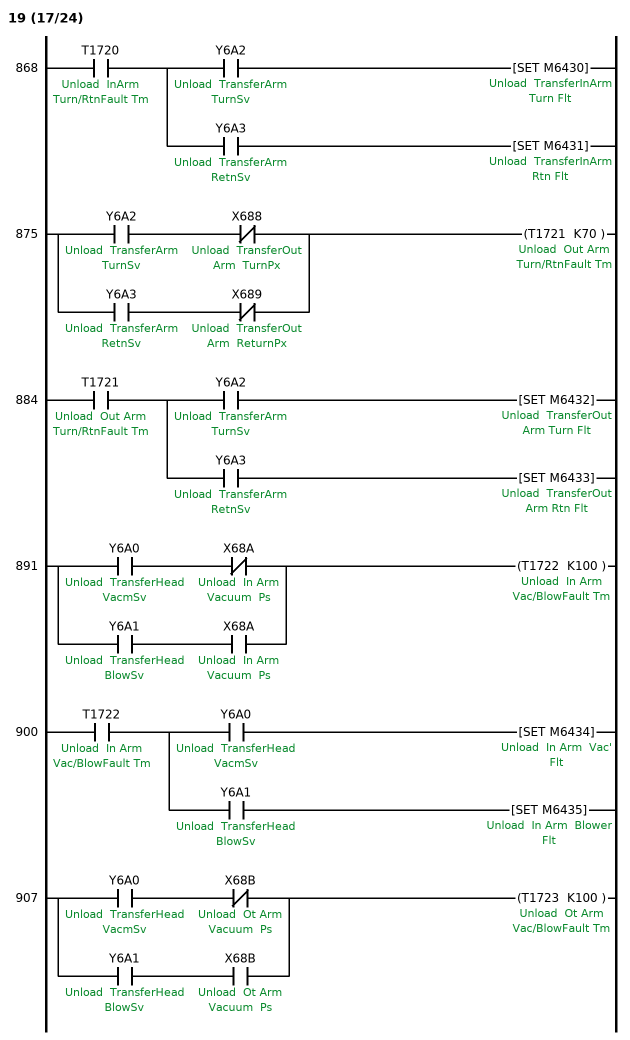
868   LD      T1720  ; Unload  InArm   Turn/RtnFault Tm
      MPS
      AND     Y6A2  ; Unload  TransferArm TurnSv
      SET     M6430  ; Unload  TransferInArm   Turn Flt
      MPP
      AND     Y6A3  ; Unload  TransferArm RetnSv
      SET     M6431  ; Unload  TransferInArm   Rtn Flt
875   LD      Y6A2  ; Unload  TransferArm TurnSv
      ANI     X688  ; Unload  TransferOutArm  TurnPx
      LD      Y6A3  ; Unload  TransferArm RetnSv
      ANI     X689  ; Unload  TransferOutArm  ReturnPx
      ORB
      OUT     T1721 K70  ; Unload  Out Arm Turn/RtnFault Tm
884   LD      T1721  ; Unload  Out Arm Turn/RtnFault Tm
      MPS
      AND     Y6A2  ; Unload  TransferArm TurnSv
      SET     M6432  ; Unload  TransferOut Arm Turn Flt
      MPP
      AND     Y6A3  ; Unload  TransferArm RetnSv
      SET     M6433  ; Unload  TransferOut Arm Rtn Flt
891   LD      Y6A0  ; Unload  TransferHeadVacmSv
      ANI     X68A  ; Unload  In Arm  Vacuum  Ps
      LD      Y6A1  ; Unload  TransferHeadBlowSv
      AND     X68A  ; Unload  In Arm  Vacuum  Ps
      ORB
      OUT     T1722 K100  ; Unload  In Arm  Vac/BlowFault Tm
900   LD      T1722  ; Unload  In Arm  Vac/BlowFault Tm
      MPS
      AND     Y6A0  ; Unload  TransferHeadVacmSv
      SET     M6434  ; Unload  In Arm  Vac' Flt
      MPP
      AND     Y6A1  ; Unload  TransferHeadBlowSv
      SET     M6435  ; Unload  In Arm  Blower  Flt
907   LD      Y6A0  ; Unload  TransferHeadVacmSv
      ANI     X68B  ; Unload  Ot Arm  Vacuum  Ps
      LD      Y6A1  ; Unload  TransferHeadBlowSv
      AND     X68B  ; Unload  Ot Arm  Vacuum  Ps
      ORB
      OUT     T1723 K100  ; Unload  Ot Arm  Vac/BlowFault Tm
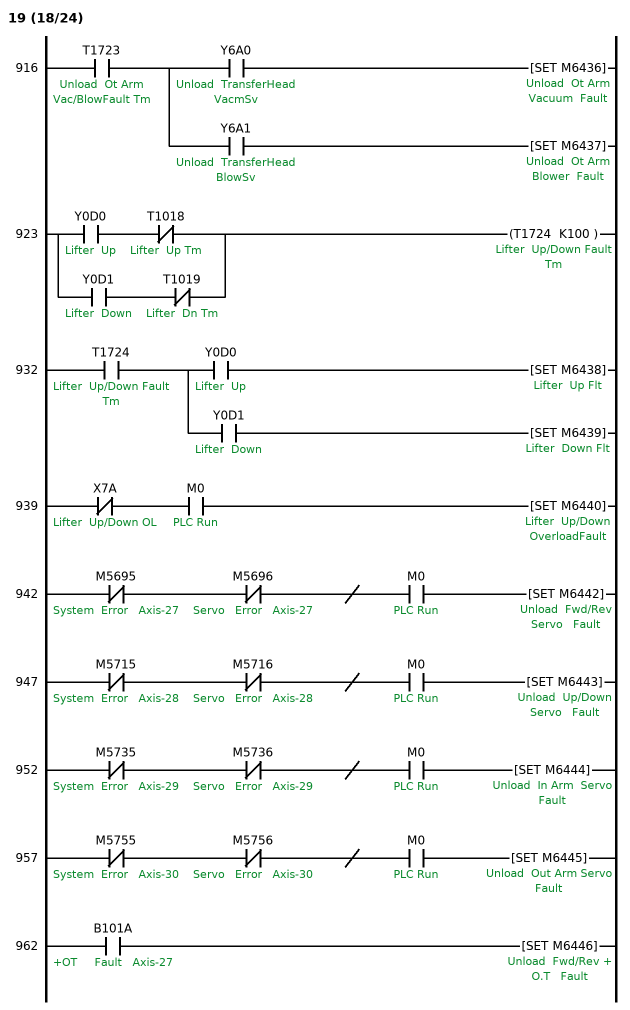
916   LD      T1723  ; Unload  Ot Arm  Vac/BlowFault Tm
      MPS
      AND     Y6A0  ; Unload  TransferHeadVacmSv
      SET     M6436  ; Unload  Ot Arm  Vacuum  Fault
      MPP
      AND     Y6A1  ; Unload  TransferHeadBlowSv
      SET     M6437  ; Unload  Ot Arm  Blower  Fault
923   LD      Y0D0  ; Lifter  Up
      ANI     T1018  ; Lifter  Up Tm
      LD      Y0D1  ; Lifter  Down
      ANI     T1019  ; Lifter  Dn Tm
      ORB
      OUT     T1724 K100  ; Lifter  Up/Down Fault Tm
932   LD      T1724  ; Lifter  Up/Down Fault Tm
      MPS
      AND     Y0D0  ; Lifter  Up
      SET     M6438  ; Lifter  Up Flt
      MPP
      AND     Y0D1  ; Lifter  Down
      SET     M6439  ; Lifter  Down Flt
939   LDI     X7A  ; Lifter  Up/Down OL
      AND     M0  ; PLC Run
      SET     M6440  ; Lifter  Up/Down OverloadFault
942   LDI     M5695  ; System  Error   Axis-27
      ANI     M5696  ; Servo   Error   Axis-27
      INV
      AND     M0  ; PLC Run
      SET     M6442  ; Unload  Fwd/Rev Servo   Fault
947   LDI     M5715  ; System  Error   Axis-28
      ANI     M5716  ; Servo   Error   Axis-28
      INV
      AND     M0  ; PLC Run
      SET     M6443  ; Unload  Up/Down Servo   Fault
952   LDI     M5735  ; System  Error   Axis-29
      ANI     M5736  ; Servo   Error   Axis-29
      INV
      AND     M0  ; PLC Run
      SET     M6444  ; Unload  In Arm  Servo   Fault
957   LDI     M5755  ; System  Error   Axis-30
      ANI     M5756  ; Servo   Error   Axis-30
      INV
      AND     M0  ; PLC Run
      SET     M6445  ; Unload  Out Arm Servo   Fault
962   LD      B101A  ; +OT     Fault   Axis-27
      SET     M6446  ; Unload  Fwd/Rev + O.T   Fault
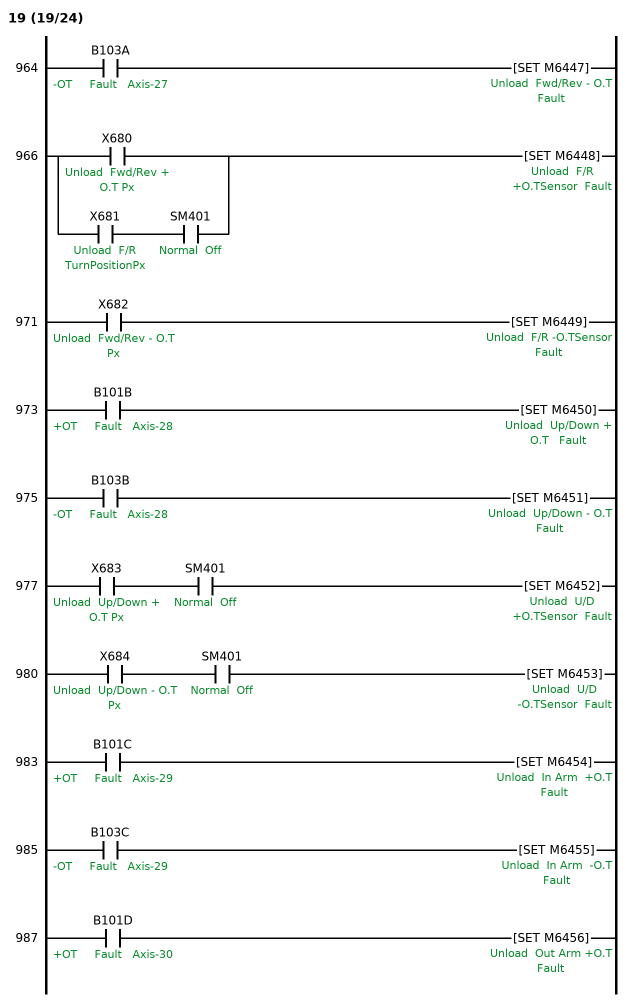
964   LD      B103A  ; -OT     Fault   Axis-27
      SET     M6447  ; Unload  Fwd/Rev - O.T   Fault
966   LD      X680  ; Unload  Fwd/Rev + O.T Px
      LD      X681  ; Unload  F/R TurnPositionPx
      AND     SM401  ; Normal  Off
      ORB
      SET     M6448  ; Unload  F/R +O.TSensor  Fault
971   LD      X682  ; Unload  Fwd/Rev - O.T Px
      SET     M6449  ; Unload  F/R -O.TSensor  Fault
973   LD      B101B  ; +OT     Fault   Axis-28
      SET     M6450  ; Unload  Up/Down + O.T   Fault
975   LD      B103B  ; -OT     Fault   Axis-28
      SET     M6451  ; Unload  Up/Down - O.T   Fault
977   LD      X683  ; Unload  Up/Down + O.T Px
      AND     SM401  ; Normal  Off
      SET     M6452  ; Unload  U/D +O.TSensor  Fault
980   LD      X684  ; Unload  Up/Down - O.T Px
      AND     SM401  ; Normal  Off
      SET     M6453  ; Unload  U/D -O.TSensor  Fault
983   LD      B101C  ; +OT     Fault   Axis-29
      SET     M6454  ; Unload  In Arm  +O.T    Fault
985   LD      B103C  ; -OT     Fault   Axis-29
      SET     M6455  ; Unload  In Arm  -O.T    Fault
987   LD      B101D  ; +OT     Fault   Axis-30
      SET     M6456  ; Unload  Out Arm +O.T    Fault
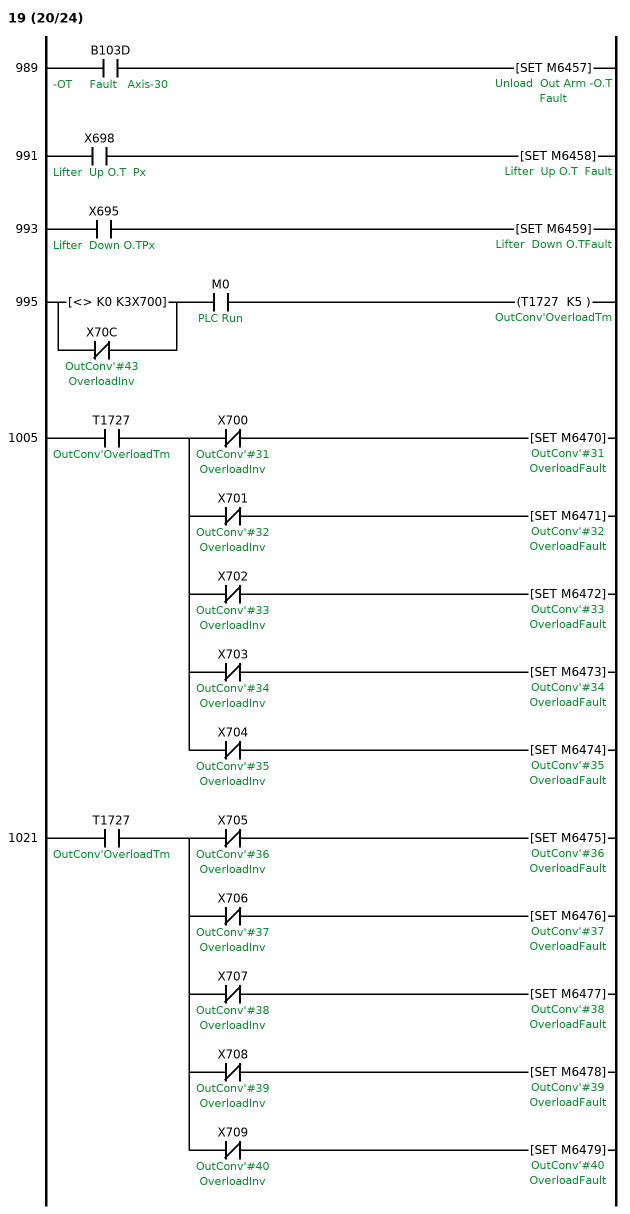
989   LD      B103D  ; -OT     Fault   Axis-30
      SET     M6457  ; Unload  Out Arm -O.T    Fault
991   LD      X698  ; Lifter  Up O.T  Px
      SET     M6458  ; Lifter  Up O.T  Fault
993   LD      X695  ; Lifter  Down O.TPx
      SET     M6459  ; Lifter  Down O.TFault
995   LD<>    K0 K3X700  ; OutConv'#31     OverloadInv
      ORI     X70C  ; OutConv'#43     OverloadInv
      AND     M0  ; PLC Run
      OUT     T1727 K5  ; OutConv'OverloadTm
1005  LD      T1727  ; OutConv'OverloadTm
      MPS
      ANI     X700  ; OutConv'#31     OverloadInv
      SET     M6470  ; OutConv'#31     OverloadFault
      MRD
      ANI     X701  ; OutConv'#32     OverloadInv
      SET     M6471  ; OutConv'#32     OverloadFault
      MRD
      ANI     X702  ; OutConv'#33     OverloadInv
      SET     M6472  ; OutConv'#33     OverloadFault
      MRD
      ANI     X703  ; OutConv'#34     OverloadInv
      SET     M6473  ; OutConv'#34     OverloadFault
      MPP
      ANI     X704  ; OutConv'#35     OverloadInv
      SET     M6474  ; OutConv'#35     OverloadFault
1021  LD      T1727  ; OutConv'OverloadTm
      MPS
      ANI     X705  ; OutConv'#36     OverloadInv
      SET     M6475  ; OutConv'#36     OverloadFault
      MRD
      ANI     X706  ; OutConv'#37     OverloadInv
      SET     M6476  ; OutConv'#37     OverloadFault
      MRD
      ANI     X707  ; OutConv'#38     OverloadInv
      SET     M6477  ; OutConv'#38     OverloadFault
      MRD
      ANI     X708  ; OutConv'#39     OverloadInv
      SET     M6478  ; OutConv'#39     OverloadFault
      MPP
      ANI     X709  ; OutConv'#40     OverloadInv
      SET     M6479  ; OutConv'#40     OverloadFault
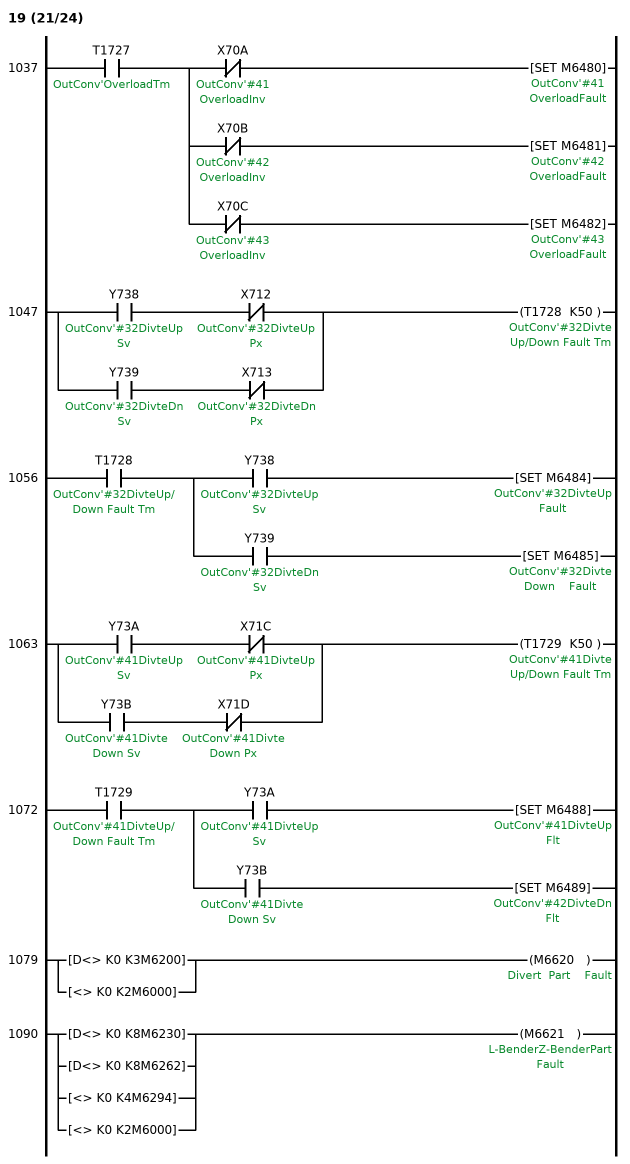
1037  LD      T1727  ; OutConv'OverloadTm
      MPS
      ANI     X70A  ; OutConv'#41     OverloadInv
      SET     M6480  ; OutConv'#41     OverloadFault
      MRD
      ANI     X70B  ; OutConv'#42     OverloadInv
      SET     M6481  ; OutConv'#42     OverloadFault
      MPP
      ANI     X70C  ; OutConv'#43     OverloadInv
      SET     M6482  ; OutConv'#43     OverloadFault
1047  LD      Y738  ; OutConv'#32DivteUp Sv
      ANI     X712  ; OutConv'#32DivteUp Px
      LD      Y739  ; OutConv'#32DivteDn Sv
      ANI     X713  ; OutConv'#32DivteDn Px
      ORB
      OUT     T1728 K50  ; OutConv'#32DivteUp/Down Fault Tm
1056  LD      T1728  ; OutConv'#32DivteUp/Down Fault Tm
      MPS
      AND     Y738  ; OutConv'#32DivteUp Sv
      SET     M6484  ; OutConv'#32DivteUp Fault
      MPP
      AND     Y739  ; OutConv'#32DivteDn Sv
      SET     M6485  ; OutConv'#32DivteDown    Fault
1063  LD      Y73A  ; OutConv'#41DivteUp Sv
      ANI     X71C  ; OutConv'#41DivteUp Px
      LD      Y73B  ; OutConv'#41DivteDown Sv
      ANI     X71D  ; OutConv'#41DivteDown Px
      ORB
      OUT     T1729 K50  ; OutConv'#41DivteUp/Down Fault Tm
1072  LD      T1729  ; OutConv'#41DivteUp/Down Fault Tm
      MPS
      AND     Y73A  ; OutConv'#41DivteUp Sv
      SET     M6488  ; OutConv'#41DivteUp Flt
      MPP
      AND     Y73B  ; OutConv'#41DivteDown Sv
      SET     M6489  ; OutConv'#42DivteDn Flt
1079  LDD<>   K0 K3M6200  ; Divert#1In Conv'OL Fault
      OR<>    K0 K2M6000  ; Emg-StopFault
      OUT     M6620  ; Divert  Part    Fault
1090  LDD<>   K0 K8M6230  ; Z-BendInClamp UpFault
      ORD<>   K0 K8M6262  ; Z-Bend  Conv' UpFault
      OR<>    K0 K4M6294  ; Z-BendInServo   Fault
      OR<>    K0 K2M6000  ; Emg-StopFault
      OUT     M6621  ; L-BenderZ-BenderPart    Fault
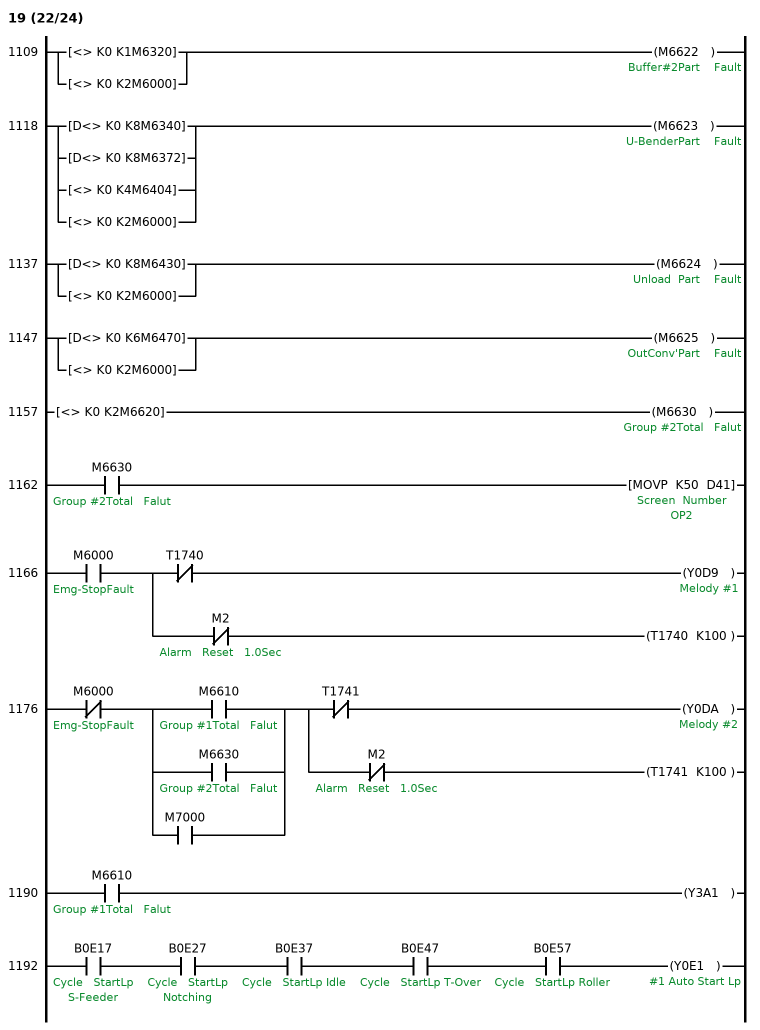
1109  LD<>    K0 K1M6320  ; Buffer#2ConveyorConv' OLFault
      OR<>    K0 K2M6000  ; Emg-StopFault
      OUT     M6622  ; Buffer#2Part    Fault
1118  LDD<>   K0 K8M6340  ; U-BenderConv' OLFalut
      ORD<>   K0 K8M6372  ; U-BendOtUpper   Guide   FwdFault
      OR<>    K0 K4M6404  ; U-BendOtLength  Unit    +O.TFlt
      OR<>    K0 K2M6000  ; Emg-StopFault
      OUT     M6623  ; U-BenderPart    Fault
1137  LDD<>   K0 K8M6430  ; Unload  TransferInArm   Turn Flt
      OR<>    K0 K2M6000  ; Emg-StopFault
      OUT     M6624  ; Unload  Part    Fault
1147  LDD<>   K0 K6M6470  ; OutConv'#31     OverloadFault
      OR<>    K0 K2M6000  ; Emg-StopFault
      OUT     M6625  ; OutConv'Part    Fault
1157  LD<>    K0 K2M6620  ; Divert  Part    Fault
      OUT     M6630  ; Group #2Total   Falut
1162  LD      M6630  ; Group #2Total   Falut
      MOVP    K50 D41  ; Screen  Number  OP2
1166  LD      M6000  ; Emg-StopFault
      MPS
      ANI     T1740
      OUT     Y0D9  ; Melody #1
      MPP
      ANI     M2  ; Alarm   Reset   1.0Sec
      OUT     T1740 K100
1176  LDI     M6000  ; Emg-StopFault
      LD      M6610  ; Group #1Total   Falut
      OR      M6630  ; Group #2Total   Falut
      OR      M7000
      ANB
      MPS
      ANI     T1741
      OUT     Y0DA  ; Melody #2
      MPP
      ANI     M2  ; Alarm   Reset   1.0Sec
      OUT     T1741 K100
1190  LD      M6610  ; Group #1Total   Falut
      OUT     Y3A1
1192  LD      B0E17  ; Cycle   StartLp S-Feeder
      AND     B0E27  ; Cycle   StartLp Notching
      AND     B0E37  ; Cycle   StartLp Idle
      AND     B0E47  ; Cycle   StartLp T-Over
      AND     B0E57  ; Cycle   StartLp Roller
      OUT     Y0E1  ; #1 Auto Start Lp
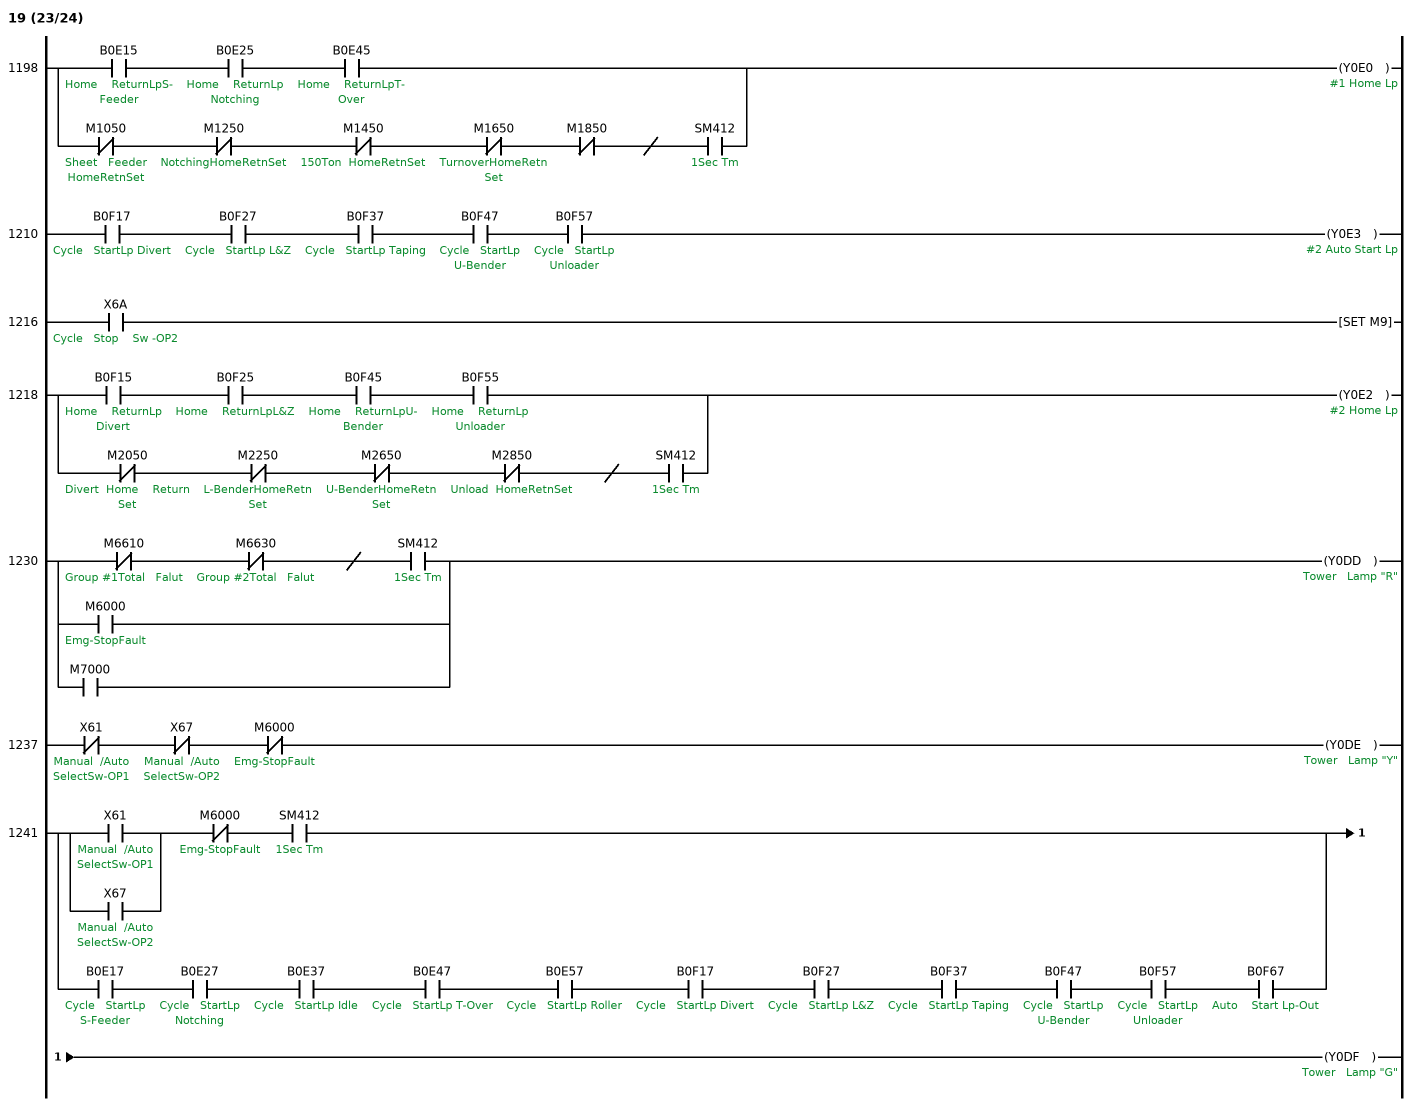
1198  LD      B0E15  ; Home    ReturnLpS-Feeder
      AND     B0E25  ; Home    ReturnLpNotching
      AND     B0E45  ; Home    ReturnLpT-Over
      LDI     M1050  ; Sheet   Feeder  HomeRetnSet
      ANI     M1250  ; NotchingHomeRetnSet
      ANI     M1450  ; 150Ton  HomeRetnSet
      ANI     M1650  ; TurnoverHomeRetnSet
      ANI     M1850
      INV
      AND     SM412  ; 1Sec Tm
      ORB
      OUT     Y0E0  ; #1 Home Lp
1210  LD      B0F17  ; Cycle   StartLp Divert
      AND     B0F27  ; Cycle   StartLp L&Z
      AND     B0F37  ; Cycle   StartLp Taping
      AND     B0F47  ; Cycle   StartLp U-Bender
      AND     B0F57  ; Cycle   StartLp Unloader
      OUT     Y0E3  ; #2 Auto Start Lp
1216  LD      X6A  ; Cycle   Stop    Sw -OP2
      SET     M9
1218  LD      B0F15  ; Home    ReturnLpDivert
      AND     B0F25  ; Home    ReturnLpL&Z
      AND     B0F45  ; Home    ReturnLpU-Bender
      AND     B0F55  ; Home    ReturnLpUnloader
      LDI     M2050  ; Divert  Home    Return  Set
      ANI     M2250  ; L-BenderHomeRetnSet
      ANI     M2650  ; U-BenderHomeRetnSet
      ANI     M2850  ; Unload  HomeRetnSet
      INV
      AND     SM412  ; 1Sec Tm
      ORB
      OUT     Y0E2  ; #2 Home Lp
1230  LDI     M6610  ; Group #1Total   Falut
      ANI     M6630  ; Group #2Total   Falut
      INV
      AND     SM412  ; 1Sec Tm
      OR      M6000  ; Emg-StopFault
      OR      M7000
      OUT     Y0DD  ; Tower   Lamp "R"
1237  LDI     X61  ; Manual  /Auto   SelectSw-OP1
      ANI     X67  ; Manual  /Auto   SelectSw-OP2
      ANI     M6000  ; Emg-StopFault
      OUT     Y0DE  ; Tower   Lamp "Y"
1241  LD      X61  ; Manual  /Auto   SelectSw-OP1
      OR      X67  ; Manual  /Auto   SelectSw-OP2
      ANI     M6000  ; Emg-StopFault
      AND     SM412  ; 1Sec Tm
      LD      B0E17  ; Cycle   StartLp S-Feeder
      AND     B0E27  ; Cycle   StartLp Notching
      AND     B0E37  ; Cycle   StartLp Idle
      AND     B0E47  ; Cycle   StartLp T-Over
      AND     B0E57  ; Cycle   StartLp Roller
      AND     B0F17  ; Cycle   StartLp Divert
      AND     B0F27  ; Cycle   StartLp L&Z
      AND     B0F37  ; Cycle   StartLp Taping
      AND     B0F47  ; Cycle   StartLp U-Bender
      AND     B0F57  ; Cycle   StartLp Unloader
      AND     B0F67  ; Auto    Start Lp-Out
      ORB
      OUT     Y0DF  ; Tower   Lamp "G"
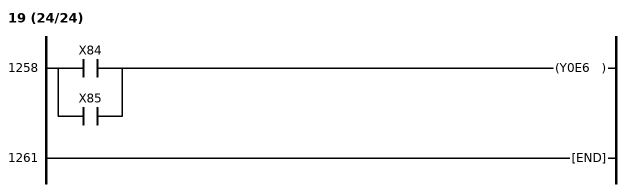
1258  LD      X84
      OR      X85
      OUT     Y0E6
1261  END
END_PROGRAM

PROGRAM 20  // #2 Conveyor Part
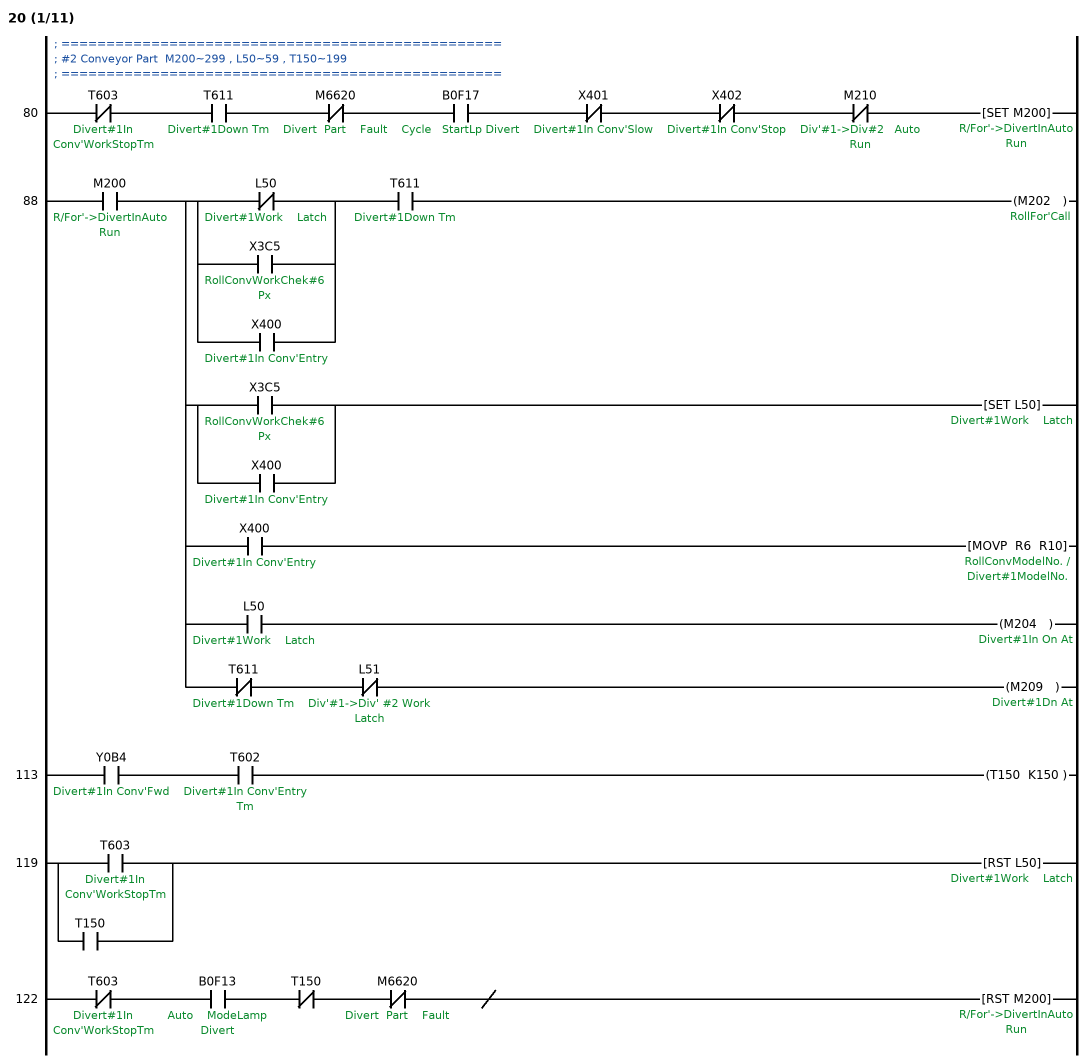
; =================================================
; #2 Conveyor Part  M200~299 , L50~59 , T150~199
; =================================================
80    LDI     T603  ; Divert#1In Conv'WorkStopTm
      AND     T611  ; Divert#1Down Tm
      ANI     M6620  ; Divert  Part    Fault
      AND     B0F17  ; Cycle   StartLp Divert
      ANI     X401  ; Divert#1In Conv'Slow
      ANI     X402  ; Divert#1In Conv'Stop
      ANI     M210  ; Div'#1->Div#2   Auto Run
      SET     M200  ; R/For'->DivertInAuto Run
88    LD      M200  ; R/For'->DivertInAuto Run
      MPS
      LDI     L50  ; Divert#1Work    Latch
      OR      X3C5  ; RollConvWorkChek#6 Px
      OR      X400  ; Divert#1In Conv'Entry
      ANB
      AND     T611  ; Divert#1Down Tm
      OUT     M202  ; RollFor'Call
      MRD
      LD      X3C5  ; RollConvWorkChek#6 Px
      OR      X400  ; Divert#1In Conv'Entry
      ANB
      SET     L50  ; Divert#1Work    Latch
      MRD
      AND     X400  ; Divert#1In Conv'Entry
      MOVP    R6 R10  ; RollConvModelNo. / Divert#1ModelNo.
      MRD
      AND     L50  ; Divert#1Work    Latch
      OUT     M204  ; Divert#1In On At
      MPP
      ANI     T611  ; Divert#1Down Tm
      ANI     L51  ; Div'#1->Div' #2 Work    Latch
      OUT     M209  ; Divert#1Dn At
113   LD      Y0B4  ; Divert#1In Conv'Fwd
      AND     T602  ; Divert#1In Conv'Entry Tm
      OUT     T150 K150
119   LD      T603  ; Divert#1In Conv'WorkStopTm
      OR      T150
      RST     L50  ; Divert#1Work    Latch
122   LDI     T603  ; Divert#1In Conv'WorkStopTm
      AND     B0F13  ; Auto    ModeLampDivert
      ANI     T150
      ANI     M6620  ; Divert  Part    Fault
      INV
      RST     M200  ; R/For'->DivertInAuto Run
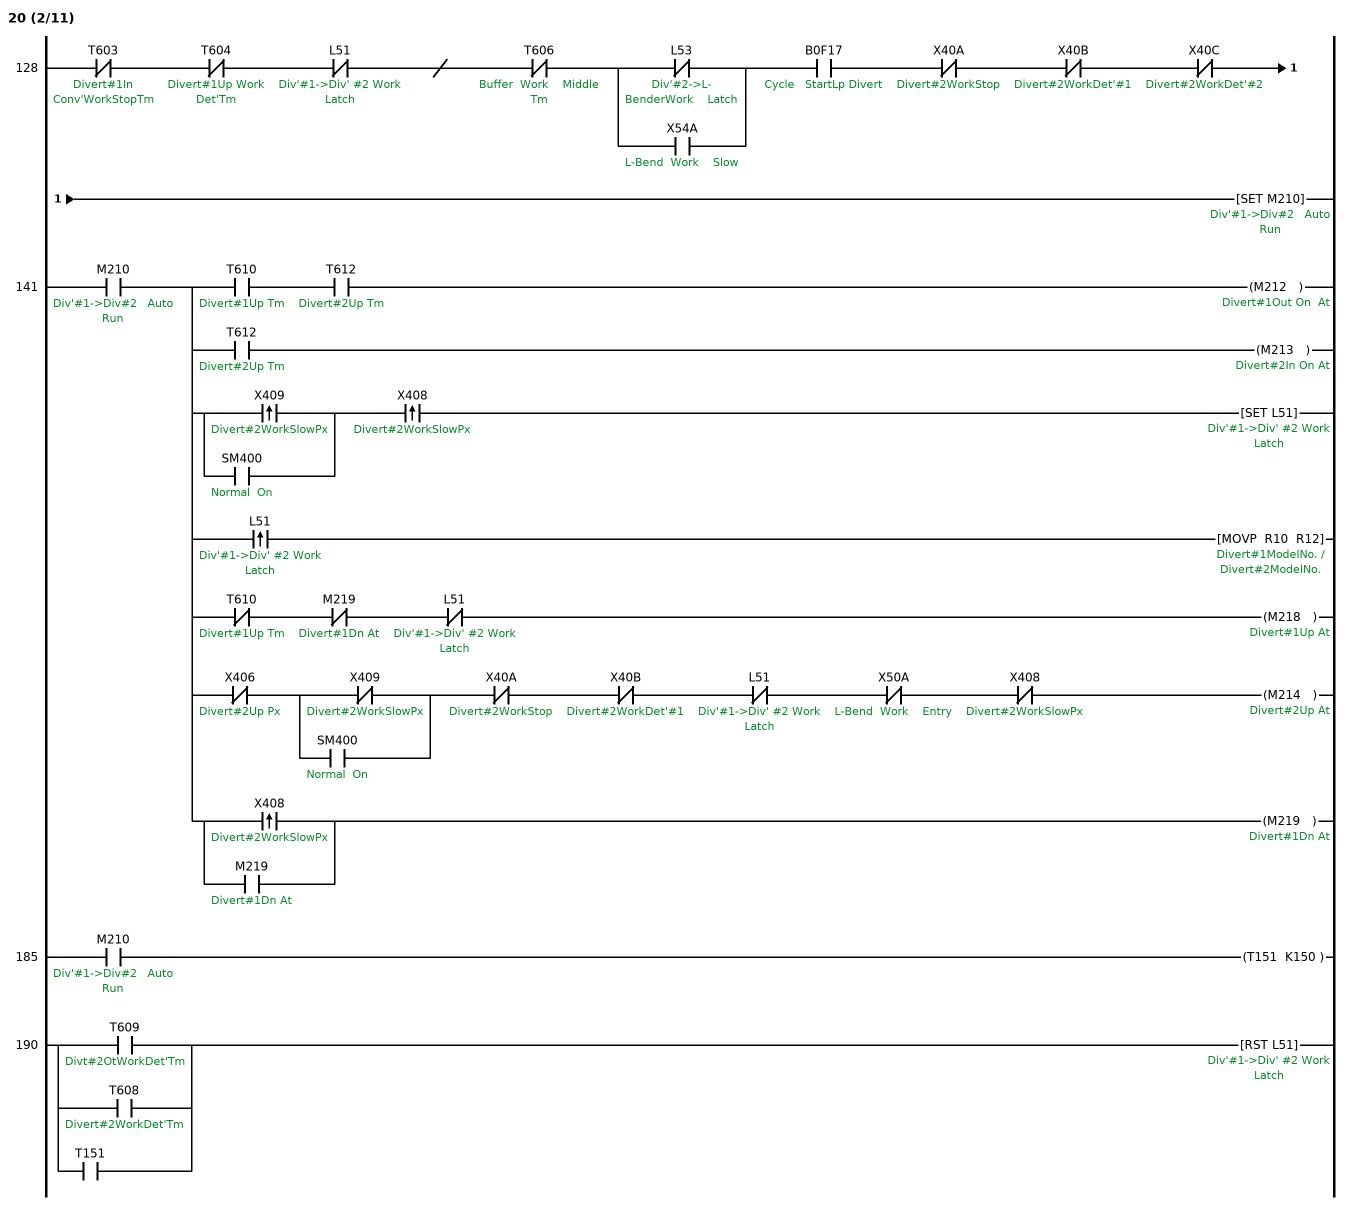
128   LDI     T603  ; Divert#1In Conv'WorkStopTm
      ANI     T604  ; Divert#1Up Work Det'Tm
      ANI     L51  ; Div'#1->Div' #2 Work    Latch
      INV
      ANI     T606  ; Buffer  Work    Middle  Tm
      LDI     L53  ; Div'#2->L-BenderWork    Latch
      OR      X54A  ; L-Bend  Work    Slow
      ANB
      AND     B0F17  ; Cycle   StartLp Divert
      ANI     X40A  ; Divert#2WorkStop
      ANI     X40B  ; Divert#2WorkDet'#1
      ANI     X40C  ; Divert#2WorkDet'#2
      SET     M210  ; Div'#1->Div#2   Auto Run
141   LD      M210  ; Div'#1->Div#2   Auto Run
      MPS
      AND     T610  ; Divert#1Up Tm
      AND     T612  ; Divert#2Up Tm
      OUT     M212  ; Divert#1Out On  At
      MRD
      AND     T612  ; Divert#2Up Tm
      OUT     M213  ; Divert#2In On At
      MRD
      LDP     X409  ; Divert#2WorkSlowPx
      OR      SM400  ; Normal  On
      ANB
      ANDP    X408  ; Divert#2WorkSlowPx
      SET     L51  ; Div'#1->Div' #2 Work    Latch
      MRD
      ANDP    L51  ; Div'#1->Div' #2 Work    Latch
      MOVP    R10 R12  ; Divert#2ModelNo.
      MRD
      ANI     T610  ; Divert#1Up Tm
      ANI     M219  ; Divert#1Dn At
      ANI     L51  ; Div'#1->Div' #2 Work    Latch
      OUT     M218  ; Divert#1Up At
      MRD
      ANI     X406  ; Divert#2Up Px
      LDI     X409  ; Divert#2WorkSlowPx
      OR      SM400  ; Normal  On
      ANB
      ANI     X40A  ; Divert#2WorkStop
      ANI     X40B  ; Divert#2WorkDet'#1
      ANI     L51  ; Div'#1->Div' #2 Work    Latch
      ANI     X50A  ; L-Bend  Work    Entry
      ANI     X408  ; Divert#2WorkSlowPx
      OUT     M214  ; Divert#2Up At
      MPP
      LDP     X408  ; Divert#2WorkSlowPx
      OR      M219  ; Divert#1Dn At
      ANB
      OUT     M219  ; Divert#1Dn At
185   LD      M210  ; Div'#1->Div#2   Auto Run
      OUT     T151 K150
190   LD      T609  ; Divt#2OtWorkDet'Tm
      OR      T608  ; Divert#2WorkDet'Tm
      OR      T151
      RST     L51  ; Div'#1->Div' #2 Work    Latch
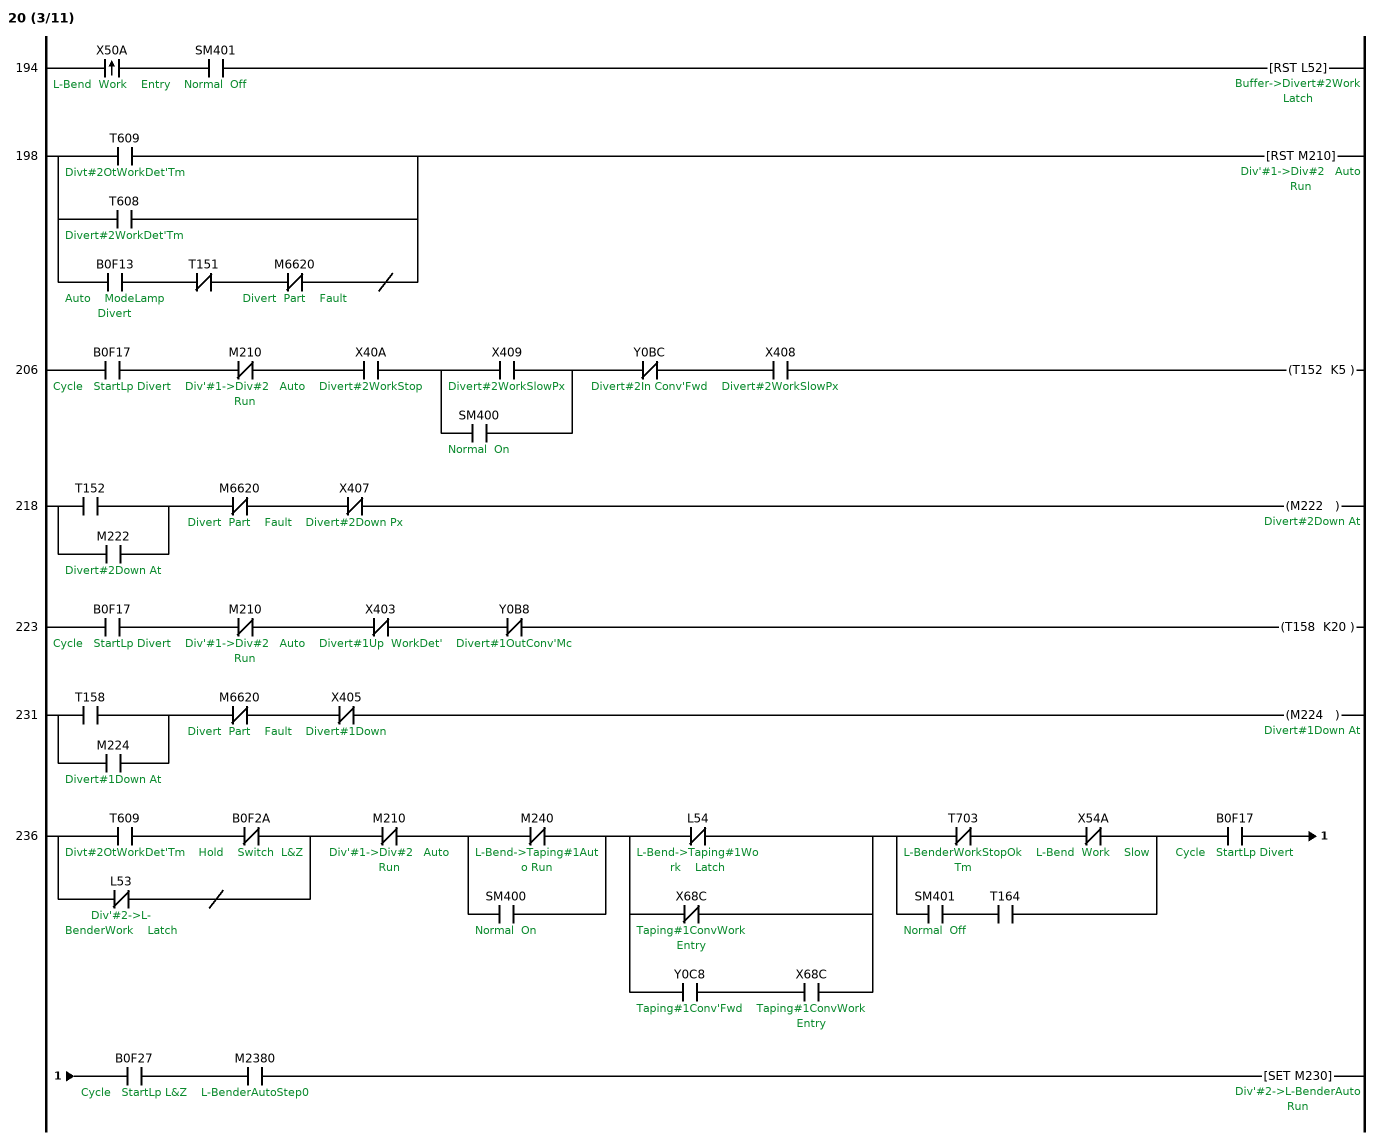
194   LDP     X50A  ; L-Bend  Work    Entry
      AND     SM401  ; Normal  Off
      RST     L52  ; Buffer->Divert#2Work    Latch
198   LD      T609  ; Divt#2OtWorkDet'Tm
      OR      T608  ; Divert#2WorkDet'Tm
      LD      B0F13  ; Auto    ModeLampDivert
      ANI     T151
      ANI     M6620  ; Divert  Part    Fault
      INV
      ORB
      RST     M210  ; Div'#1->Div#2   Auto Run
206   LD      B0F17  ; Cycle   StartLp Divert
      ANI     M210  ; Div'#1->Div#2   Auto Run
      AND     X40A  ; Divert#2WorkStop
      LD      X409  ; Divert#2WorkSlowPx
      OR      SM400  ; Normal  On
      ANB
      ANI     Y0BC  ; Divert#2In Conv'Fwd
      AND     X408  ; Divert#2WorkSlowPx
      OUT     T152 K5
218   LD      T152
      OR      M222  ; Divert#2Down At
      ANI     M6620  ; Divert  Part    Fault
      ANI     X407  ; Divert#2Down Px
      OUT     M222  ; Divert#2Down At
223   LD      B0F17  ; Cycle   StartLp Divert
      ANI     M210  ; Div'#1->Div#2   Auto Run
      ANI     X403  ; Divert#1Up  WorkDet'
      ANI     Y0B8  ; Divert#1OutConv'Mc
      OUT     T158 K20
231   LD      T158
      OR      M224  ; Divert#1Down At
      ANI     M6620  ; Divert  Part    Fault
      ANI     X405  ; Divert#1Down
      OUT     M224  ; Divert#1Down At
236   LD      T609  ; Divt#2OtWorkDet'Tm
      ANI     B0F2A  ; Hold    Switch  L&Z
      LDI     L53  ; Div'#2->L-BenderWork    Latch
      INV
      ORB
      ANI     M210  ; Div'#1->Div#2   Auto Run
      LDI     M240  ; L-Bend->Taping#1Auto Run
      OR      SM400  ; Normal  On
      ANB
      LDI     L54  ; L-Bend->Taping#1Work    Latch
      ORI     X68C  ; Taping#1ConvWorkEntry
      LD      Y0C8  ; Taping#1Conv'Fwd
      AND     X68C  ; Taping#1ConvWorkEntry
      ORB
      ANB
      LDI     T703  ; L-BenderWorkStopOk Tm
      ANI     X54A  ; L-Bend  Work    Slow
      LD      SM401  ; Normal  Off
      AND     T164
      ORB
      ANB
      AND     B0F17  ; Cycle   StartLp Divert
      AND     B0F27  ; Cycle   StartLp L&Z
      AND     M2380  ; L-BenderAutoStep0
      SET     M230  ; Div'#2->L-BenderAuto Run
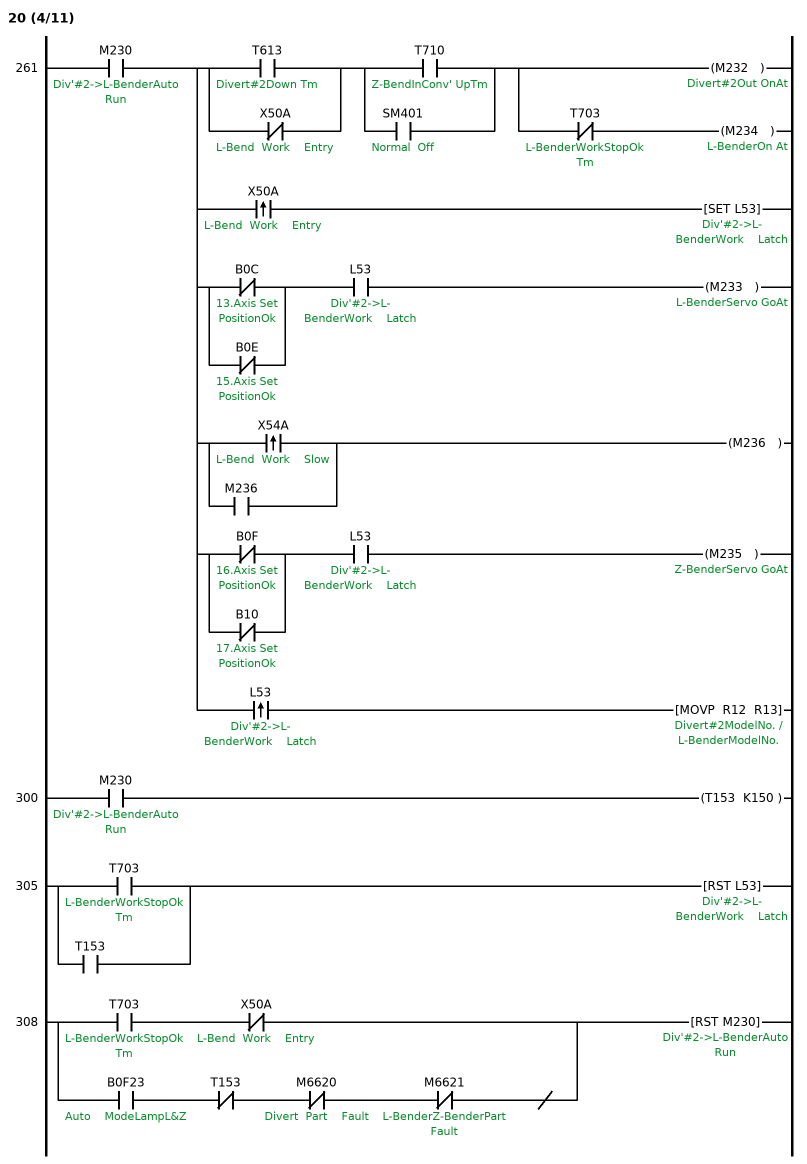
261   LD      M230  ; Div'#2->L-BenderAuto Run
      MPS
      LD      T613  ; Divert#2Down Tm
      ORI     X50A  ; L-Bend  Work    Entry
      ANB
      LD      T710  ; Z-BendInConv' UpTm
      OR      SM401  ; Normal  Off
      ANB
      OUT     M232  ; Divert#2Out OnAt
      ANI     T703  ; L-BenderWorkStopOk Tm
      OUT     M234  ; L-BenderOn At
      MRD
      ANDP    X50A  ; L-Bend  Work    Entry
      SET     L53  ; Div'#2->L-BenderWork    Latch
      MRD
      LDI     B0C  ; 13.Axis Set     PositionOk
      ORI     B0E  ; 15.Axis Set     PositionOk
      ANB
      AND     L53  ; Div'#2->L-BenderWork    Latch
      OUT     M233  ; L-BenderServo GoAt
      MRD
      LDP     X54A  ; L-Bend  Work    Slow
      OR      M236
      ANB
      OUT     M236
      MRD
      LDI     B0F  ; 16.Axis Set     PositionOk
      ORI     B10  ; 17.Axis Set     PositionOk
      ANB
      AND     L53  ; Div'#2->L-BenderWork    Latch
      OUT     M235  ; Z-BenderServo GoAt
      MPP
      ANDP    L53  ; Div'#2->L-BenderWork    Latch
      MOVP    R12 R13  ; L-BenderModelNo.
300   LD      M230  ; Div'#2->L-BenderAuto Run
      OUT     T153 K150
305   LD      T703  ; L-BenderWorkStopOk Tm
      OR      T153
      RST     L53  ; Div'#2->L-BenderWork    Latch
308   LD      T703  ; L-BenderWorkStopOk Tm
      ANI     X50A  ; L-Bend  Work    Entry
      LD      B0F23  ; Auto    ModeLampL&Z
      ANI     T153
      ANI     M6620  ; Divert  Part    Fault
      ANI     M6621  ; L-BenderZ-BenderPart    Fault
      INV
      ORB
      RST     M230  ; Div'#2->L-BenderAuto Run
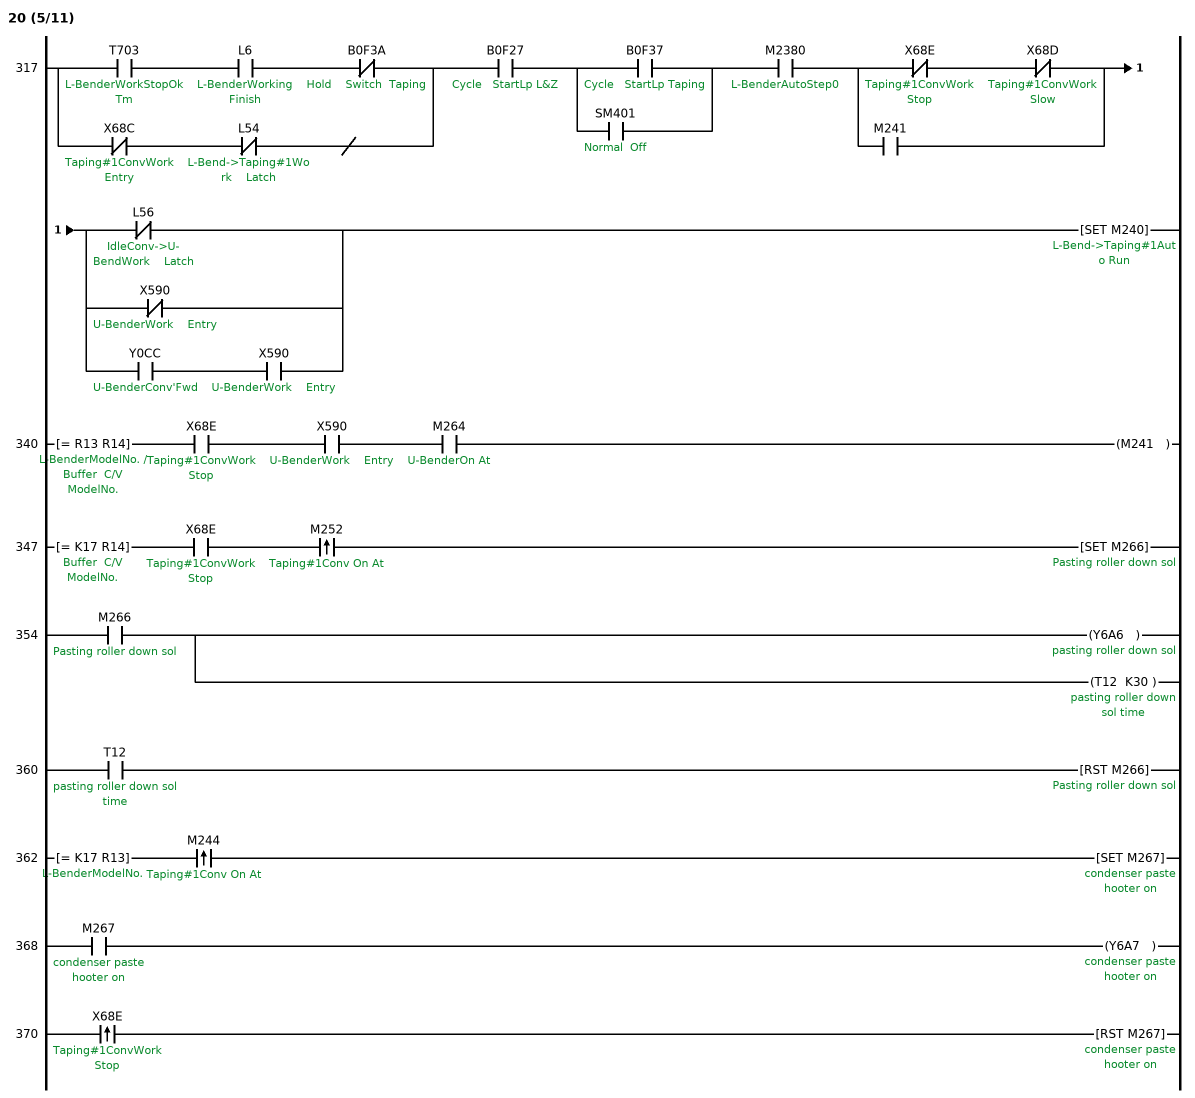
317   LD      T703  ; L-BenderWorkStopOk Tm
      AND     L6  ; L-BenderWorking Finish
      ANI     B0F3A  ; Hold    Switch  Taping
      LDI     X68C  ; Taping#1ConvWorkEntry
      ANI     L54  ; L-Bend->Taping#1Work    Latch
      INV
      ORB
      AND     B0F27  ; Cycle   StartLp L&Z
      LD      B0F37  ; Cycle   StartLp Taping
      OR      SM401  ; Normal  Off
      ANB
      AND     M2380  ; L-BenderAutoStep0
      LDI     X68E  ; Taping#1ConvWorkStop
      ANI     X68D  ; Taping#1ConvWorkSlow
      OR      M241
      ANB
      LDI     L56  ; IdleConv->U-BendWork    Latch
      ORI     X590  ; U-BenderWork    Entry
      LD      Y0CC  ; U-BenderConv'Fwd
      AND     X590  ; U-BenderWork    Entry
      ORB
      ANB
      SET     M240  ; L-Bend->Taping#1Auto Run
340   LD=     R13 R14  ; L-BenderModelNo. / Buffer  C/V     ModelNo.
      AND     X68E  ; Taping#1ConvWorkStop
      AND     X590  ; U-BenderWork    Entry
      AND     M264  ; U-BenderOn At
      OUT     M241
347   LD=     K17 R14  ; Buffer  C/V     ModelNo.
      AND     X68E  ; Taping#1ConvWorkStop
      ANDP    M252  ; Taping#1Conv On At
      SET     M266  ; Pasting roller down sol
354   LD      M266  ; Pasting roller down sol
      OUT     Y6A6  ; pasting roller down sol
      OUT     T12 K30  ; pasting roller down sol time
360   LD      T12  ; pasting roller down sol time
      RST     M266  ; Pasting roller down sol
362   LD=     K17 R13  ; L-BenderModelNo.
      ANDP    M244  ; Taping#1Conv On At
      SET     M267  ; condenser paste hooter on
368   LD      M267  ; condenser paste hooter on
      OUT     Y6A7  ; condenser paste hooter on
370   LDP     X68E  ; Taping#1ConvWorkStop
      RST     M267  ; condenser paste hooter on
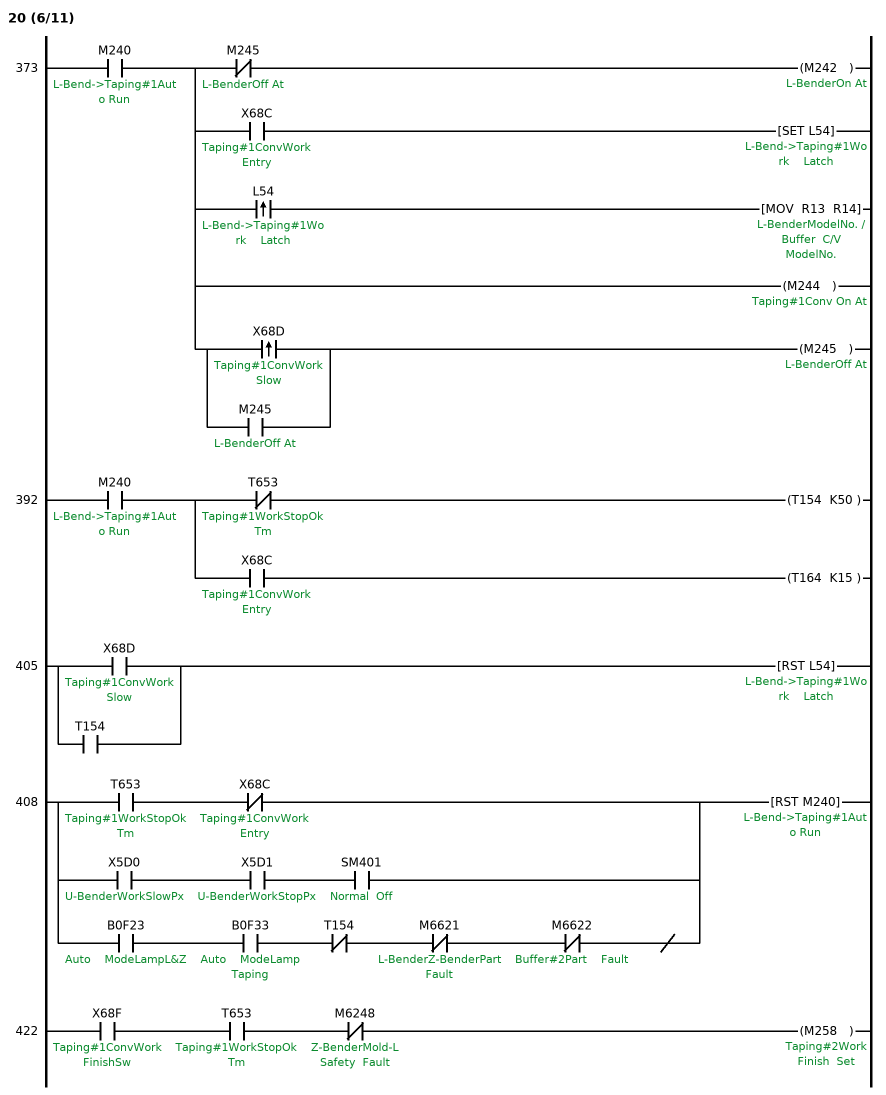
373   LD      M240  ; L-Bend->Taping#1Auto Run
      MPS
      ANI     M245  ; L-BenderOff At
      OUT     M242  ; L-BenderOn At
      MRD
      AND     X68C  ; Taping#1ConvWorkEntry
      SET     L54  ; L-Bend->Taping#1Work    Latch
      MRD
      ANDP    L54  ; L-Bend->Taping#1Work    Latch
      MOV     R13 R14
      MPP
      OUT     M244  ; Taping#1Conv On At
      LDP     X68D  ; Taping#1ConvWorkSlow
      OR      M245  ; L-BenderOff At
      ANB
      OUT     M245  ; L-BenderOff At
392   LD      M240  ; L-Bend->Taping#1Auto Run
      MPS
      ANI     T653  ; Taping#1WorkStopOk Tm
      OUT     T154 K50
      MPP
      AND     X68C  ; Taping#1ConvWorkEntry
      OUT     T164 K15
405   LD      X68D  ; Taping#1ConvWorkSlow
      OR      T154
      RST     L54  ; L-Bend->Taping#1Work    Latch
408   LD      T653  ; Taping#1WorkStopOk Tm
      ANI     X68C  ; Taping#1ConvWorkEntry
      LD      X5D0  ; U-BenderWorkSlowPx
      AND     X5D1  ; U-BenderWorkStopPx
      AND     SM401  ; Normal  Off
      ORB
      LD      B0F23  ; Auto    ModeLampL&Z
      AND     B0F33  ; Auto    ModeLampTaping
      ANI     T154
      ANI     M6621  ; L-BenderZ-BenderPart    Fault
      ANI     M6622  ; Buffer#2Part    Fault
      INV
      ORB
      RST     M240  ; L-Bend->Taping#1Auto Run
422   LD      X68F  ; Taping#1ConvWorkFinishSw
      AND     T653  ; Taping#1WorkStopOk Tm
      ANI     M6248  ; Z-BenderMold-L  Safety  Fault
      OUT     M258  ; Taping#2Work    Finish  Set
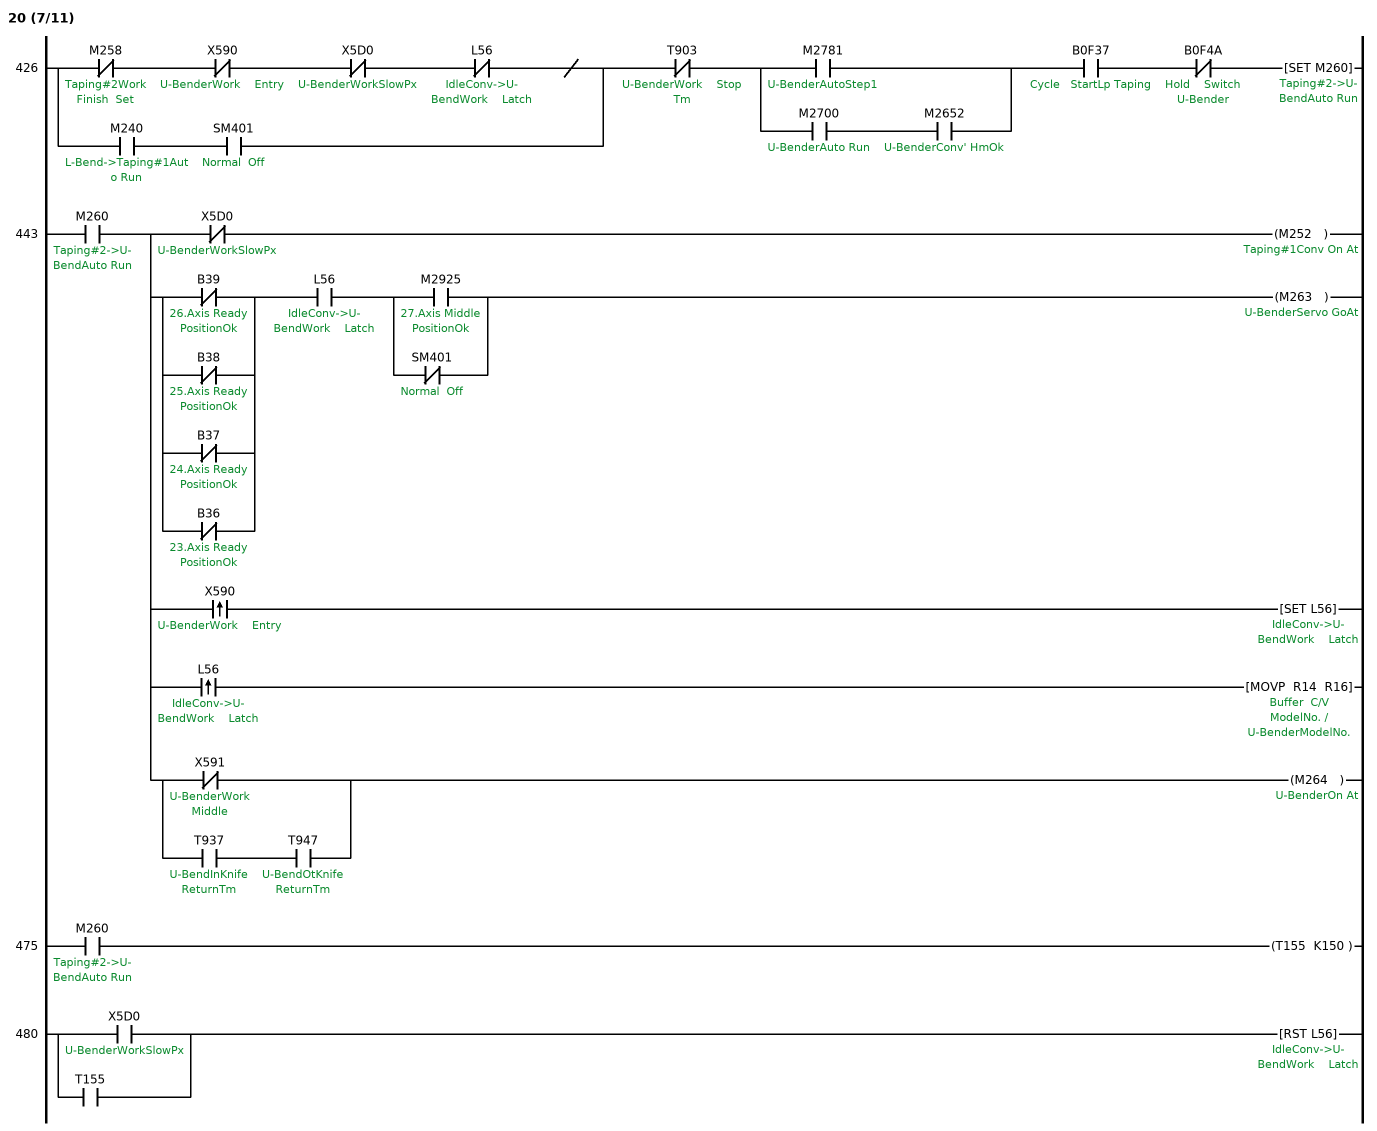
426   LDI     M258  ; Taping#2Work    Finish  Set
      ANI     X590  ; U-BenderWork    Entry
      ANI     X5D0  ; U-BenderWorkSlowPx
      ANI     L56  ; IdleConv->U-BendWork    Latch
      INV
      LD      M240  ; L-Bend->Taping#1Auto Run
      AND     SM401  ; Normal  Off
      ORB
      ANI     T903  ; U-BenderWork    Stop Tm
      LD      M2781  ; U-BenderAutoStep1
      LD      M2700  ; U-BenderAuto Run
      AND     M2652  ; U-BenderConv' HmOk
      ORB
      ANB
      AND     B0F37  ; Cycle   StartLp Taping
      ANI     B0F4A  ; Hold    Switch  U-Bender
      SET     M260  ; Taping#2->U-BendAuto Run
443   LD      M260  ; Taping#2->U-BendAuto Run
      MPS
      ANI     X5D0  ; U-BenderWorkSlowPx
      OUT     M252  ; Taping#1Conv On At
      MRD
      LDI     B39  ; 26.Axis Ready   PositionOk
      ORI     B38  ; 25.Axis Ready   PositionOk
      ORI     B37  ; 24.Axis Ready   PositionOk
      ORI     B36  ; 23.Axis Ready   PositionOk
      ANB
      AND     L56  ; IdleConv->U-BendWork    Latch
      LD      M2925  ; 27.Axis Middle  PositionOk
      ORI     SM401  ; Normal  Off
      ANB
      OUT     M263  ; U-BenderServo GoAt
      MRD
      ANDP    X590  ; U-BenderWork    Entry
      SET     L56  ; IdleConv->U-BendWork    Latch
      MRD
      ANDP    L56  ; IdleConv->U-BendWork    Latch
      MOVP    R14 R16  ; U-BenderModelNo.
      MPP
      LDI     X591  ; U-BenderWork    Middle
      LD      T937  ; U-BendInKnife   ReturnTm
      AND     T947  ; U-BendOtKnife   ReturnTm
      ORB
      ANB
      OUT     M264  ; U-BenderOn At
475   LD      M260  ; Taping#2->U-BendAuto Run
      OUT     T155 K150
480   LD      X5D0  ; U-BenderWorkSlowPx
      OR      T155
      RST     L56  ; IdleConv->U-BendWork    Latch
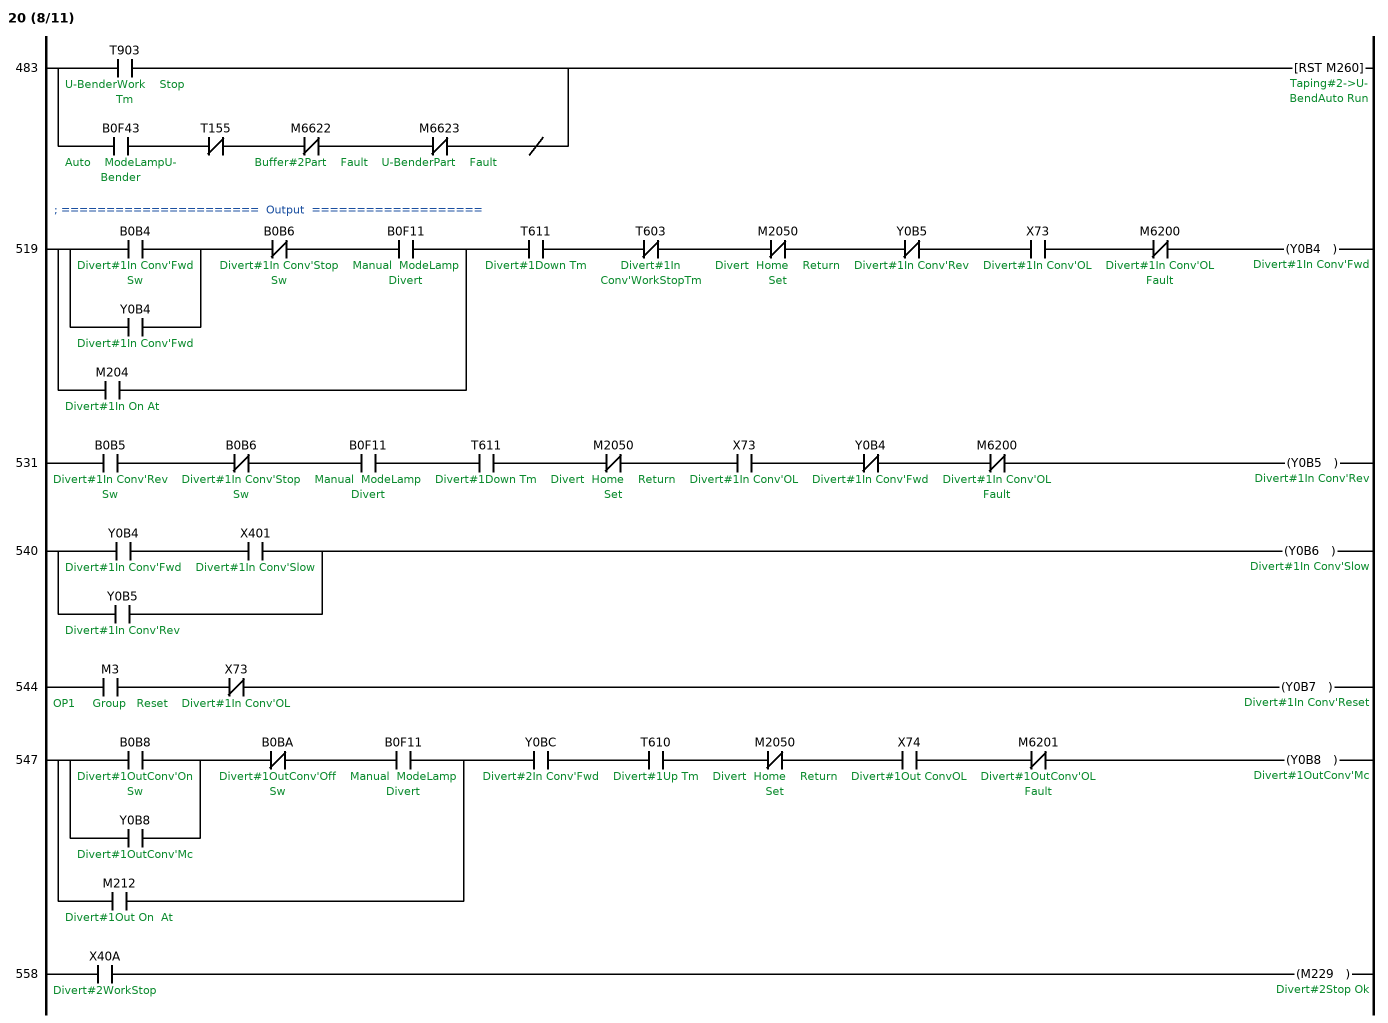
483   LD      T903  ; U-BenderWork    Stop Tm
      LD      B0F43  ; Auto    ModeLampU-Bender
      ANI     T155
      ANI     M6622  ; Buffer#2Part    Fault
      ANI     M6623  ; U-BenderPart    Fault
      INV
      ORB
      RST     M260  ; Taping#2->U-BendAuto Run
; ======================  Output  ===================
519   LD      B0B4  ; Divert#1In Conv'Fwd Sw
      OR      Y0B4  ; Divert#1In Conv'Fwd
      ANI     B0B6  ; Divert#1In Conv'Stop Sw
      AND     B0F11  ; Manual  ModeLampDivert
      OR      M204  ; Divert#1In On At
      AND     T611  ; Divert#1Down Tm
      ANI     T603  ; Divert#1In Conv'WorkStopTm
      ANI     M2050  ; Divert  Home    Return  Set
      ANI     Y0B5  ; Divert#1In Conv'Rev
      AND     X73  ; Divert#1In Conv'OL
      ANI     M6200  ; Divert#1In Conv'OL Fault
      OUT     Y0B4  ; Divert#1In Conv'Fwd
531   LD      B0B5  ; Divert#1In Conv'Rev Sw
      ANI     B0B6  ; Divert#1In Conv'Stop Sw
      AND     B0F11  ; Manual  ModeLampDivert
      AND     T611  ; Divert#1Down Tm
      ANI     M2050  ; Divert  Home    Return  Set
      AND     X73  ; Divert#1In Conv'OL
      ANI     Y0B4  ; Divert#1In Conv'Fwd
      ANI     M6200  ; Divert#1In Conv'OL Fault
      OUT     Y0B5  ; Divert#1In Conv'Rev
540   LD      Y0B4  ; Divert#1In Conv'Fwd
      AND     X401  ; Divert#1In Conv'Slow
      OR      Y0B5  ; Divert#1In Conv'Rev
      OUT     Y0B6  ; Divert#1In Conv'Slow
544   LD      M3  ; OP1     Group   Reset
      ANI     X73  ; Divert#1In Conv'OL
      OUT     Y0B7  ; Divert#1In Conv'Reset
547   LD      B0B8  ; Divert#1OutConv'On Sw
      OR      Y0B8  ; Divert#1OutConv'Mc
      ANI     B0BA  ; Divert#1OutConv'OffSw
      AND     B0F11  ; Manual  ModeLampDivert
      OR      M212  ; Divert#1Out On  At
      AND     Y0BC  ; Divert#2In Conv'Fwd
      AND     T610  ; Divert#1Up Tm
      ANI     M2050  ; Divert  Home    Return  Set
      AND     X74  ; Divert#1Out ConvOL
      ANI     M6201  ; Divert#1OutConv'OL Fault
      OUT     Y0B8  ; Divert#1OutConv'Mc
558   LD      X40A  ; Divert#2WorkStop
      OUT     M229  ; Divert#2Stop Ok
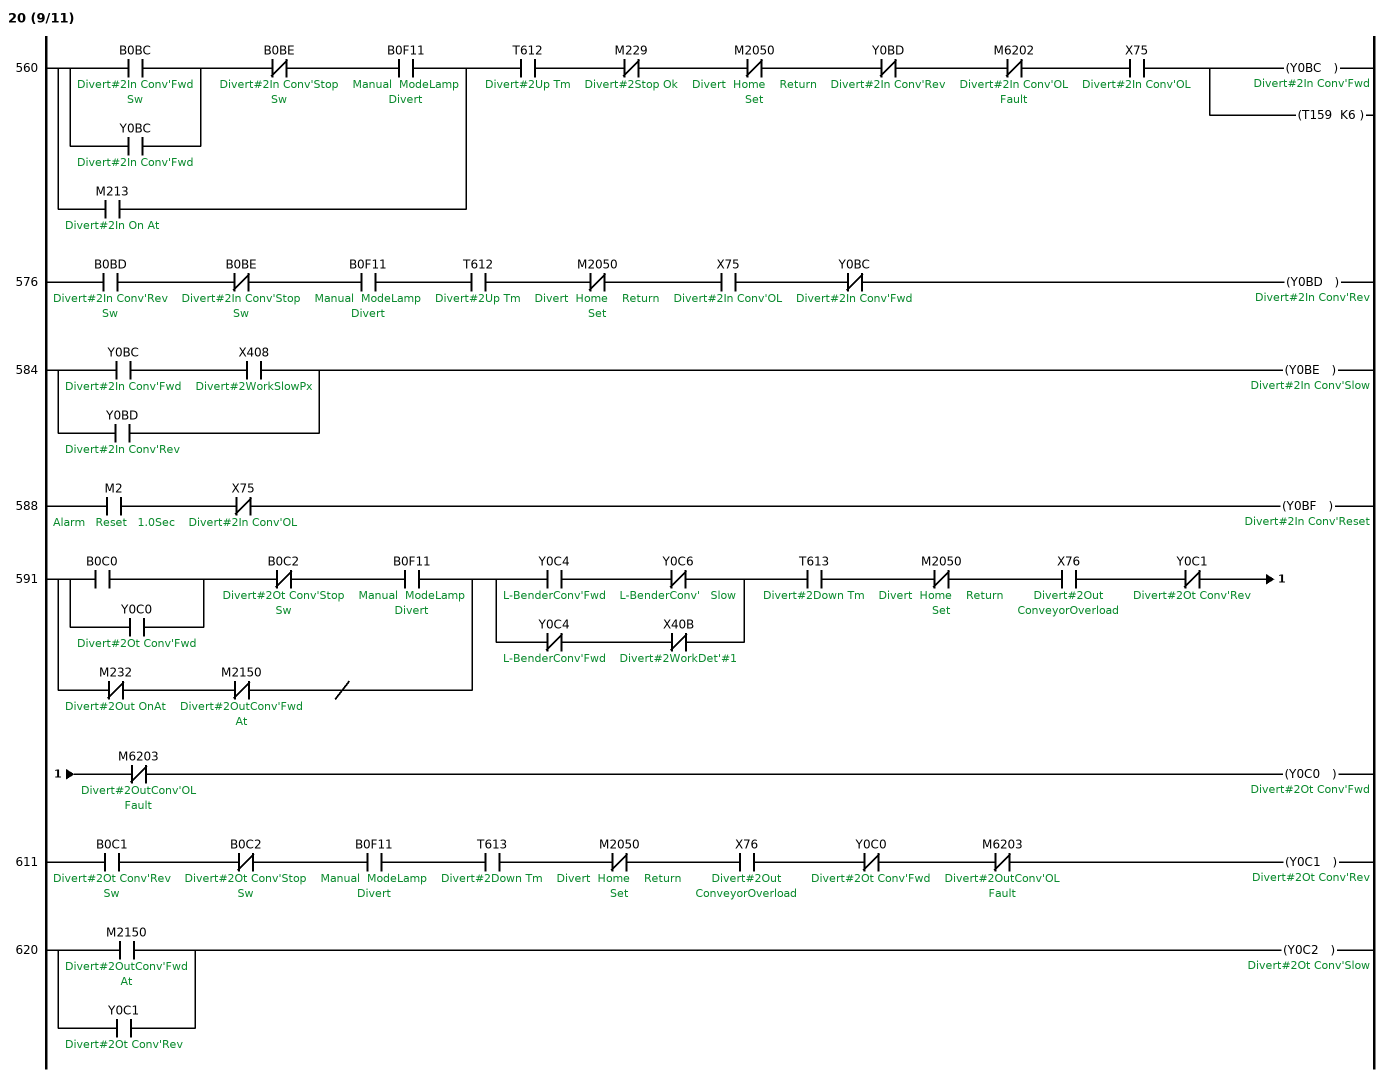
560   LD      B0BC  ; Divert#2In Conv'Fwd Sw
      OR      Y0BC  ; Divert#2In Conv'Fwd
      ANI     B0BE  ; Divert#2In Conv'Stop Sw
      AND     B0F11  ; Manual  ModeLampDivert
      OR      M213  ; Divert#2In On At
      AND     T612  ; Divert#2Up Tm
      ANI     M229  ; Divert#2Stop Ok
      ANI     M2050  ; Divert  Home    Return  Set
      ANI     Y0BD  ; Divert#2In Conv'Rev
      ANI     M6202  ; Divert#2In Conv'OL Fault
      AND     X75  ; Divert#2In Conv'OL
      OUT     Y0BC  ; Divert#2In Conv'Fwd
      OUT     T159 K6
576   LD      B0BD  ; Divert#2In Conv'Rev Sw
      ANI     B0BE  ; Divert#2In Conv'Stop Sw
      AND     B0F11  ; Manual  ModeLampDivert
      AND     T612  ; Divert#2Up Tm
      ANI     M2050  ; Divert  Home    Return  Set
      AND     X75  ; Divert#2In Conv'OL
      ANI     Y0BC  ; Divert#2In Conv'Fwd
      OUT     Y0BD  ; Divert#2In Conv'Rev
584   LD      Y0BC  ; Divert#2In Conv'Fwd
      AND     X408  ; Divert#2WorkSlowPx
      OR      Y0BD  ; Divert#2In Conv'Rev
      OUT     Y0BE  ; Divert#2In Conv'Slow
588   LD      M2  ; Alarm   Reset   1.0Sec
      ANI     X75  ; Divert#2In Conv'OL
      OUT     Y0BF  ; Divert#2In Conv'Reset
591   LD      B0C0
      OR      Y0C0  ; Divert#2Ot Conv'Fwd
      ANI     B0C2  ; Divert#2Ot Conv'Stop Sw
      AND     B0F11  ; Manual  ModeLampDivert
      LDI     M232  ; Divert#2Out OnAt
      ANI     M2150  ; Divert#2OutConv'FwdAt
      INV
      ORB
      LD      Y0C4  ; L-BenderConv'Fwd
      ANI     Y0C6  ; L-BenderConv'   Slow
      LDI     Y0C4  ; L-BenderConv'Fwd
      ANI     X40B  ; Divert#2WorkDet'#1
      ORB
      ANB
      AND     T613  ; Divert#2Down Tm
      ANI     M2050  ; Divert  Home    Return  Set
      AND     X76  ; Divert#2Out     ConveyorOverload
      ANI     Y0C1  ; Divert#2Ot Conv'Rev
      ANI     M6203  ; Divert#2OutConv'OL Fault
      OUT     Y0C0  ; Divert#2Ot Conv'Fwd
611   LD      B0C1  ; Divert#2Ot Conv'Rev Sw
      ANI     B0C2  ; Divert#2Ot Conv'Stop Sw
      AND     B0F11  ; Manual  ModeLampDivert
      AND     T613  ; Divert#2Down Tm
      ANI     M2050  ; Divert  Home    Return  Set
      AND     X76  ; Divert#2Out     ConveyorOverload
      ANI     Y0C0  ; Divert#2Ot Conv'Fwd
      ANI     M6203  ; Divert#2OutConv'OL Fault
      OUT     Y0C1  ; Divert#2Ot Conv'Rev
620   LD      M2150  ; Divert#2OutConv'FwdAt
      OR      Y0C1  ; Divert#2Ot Conv'Rev
      OUT     Y0C2  ; Divert#2Ot Conv'Slow
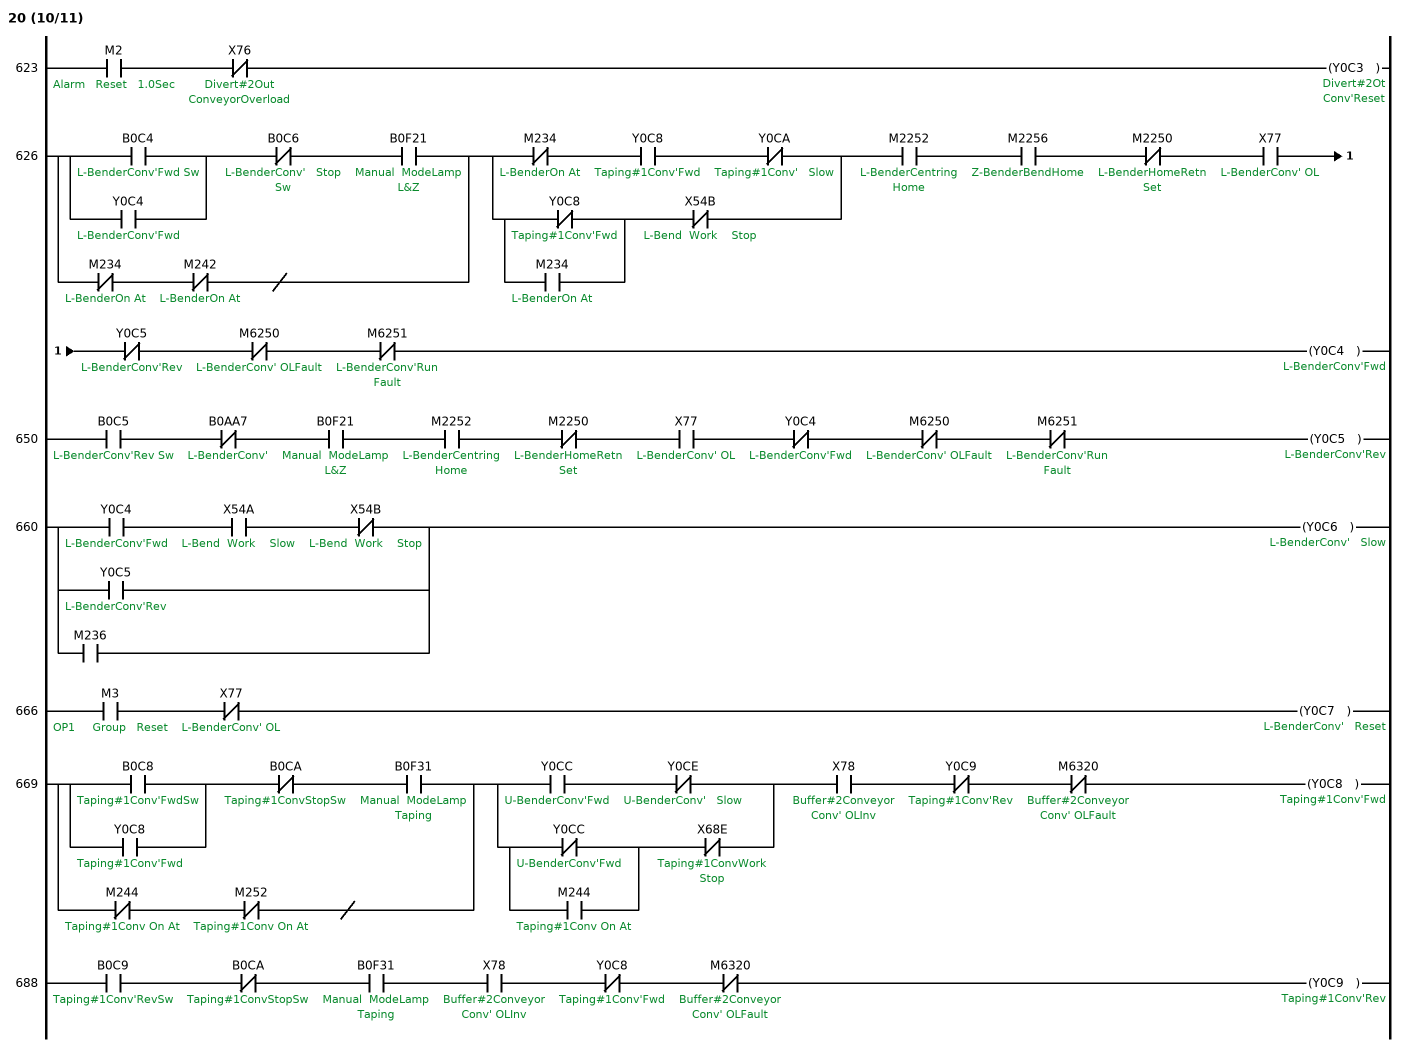
623   LD      M2  ; Alarm   Reset   1.0Sec
      ANI     X76  ; Divert#2Out     ConveyorOverload
      OUT     Y0C3  ; Divert#2Ot Conv'Reset
626   LD      B0C4  ; L-BenderConv'Fwd Sw
      OR      Y0C4  ; L-BenderConv'Fwd
      ANI     B0C6  ; L-BenderConv'   Stop Sw
      AND     B0F21  ; Manual  ModeLampL&Z
      LDI     M234  ; L-BenderOn At
      ANI     M242  ; L-BenderOn At
      INV
      ORB
      LDI     M234  ; L-BenderOn At
      AND     Y0C8  ; Taping#1Conv'Fwd
      ANI     Y0CA  ; Taping#1Conv'   Slow
      LDI     Y0C8  ; Taping#1Conv'Fwd
      OR      M234  ; L-BenderOn At
      ANI     X54B  ; L-Bend  Work    Stop
      ORB
      ANB
      AND     M2252  ; L-BenderCentringHome
      AND     M2256  ; Z-BenderBendHome
      ANI     M2250  ; L-BenderHomeRetnSet
      AND     X77  ; L-BenderConv' OL
      ANI     Y0C5  ; L-BenderConv'Rev
      ANI     M6250  ; L-BenderConv' OLFault
      ANI     M6251  ; L-BenderConv'RunFault
      OUT     Y0C4  ; L-BenderConv'Fwd
650   LD      B0C5  ; L-BenderConv'Rev Sw
      ANI     B0AA7  ; L-BenderConv'
      AND     B0F21  ; Manual  ModeLampL&Z
      AND     M2252  ; L-BenderCentringHome
      ANI     M2250  ; L-BenderHomeRetnSet
      AND     X77  ; L-BenderConv' OL
      ANI     Y0C4  ; L-BenderConv'Fwd
      ANI     M6250  ; L-BenderConv' OLFault
      ANI     M6251  ; L-BenderConv'RunFault
      OUT     Y0C5  ; L-BenderConv'Rev
660   LD      Y0C4  ; L-BenderConv'Fwd
      AND     X54A  ; L-Bend  Work    Slow
      ANI     X54B  ; L-Bend  Work    Stop
      OR      Y0C5  ; L-BenderConv'Rev
      OR      M236
      OUT     Y0C6  ; L-BenderConv'   Slow
666   LD      M3  ; OP1     Group   Reset
      ANI     X77  ; L-BenderConv' OL
      OUT     Y0C7  ; L-BenderConv'   Reset
669   LD      B0C8  ; Taping#1Conv'FwdSw
      OR      Y0C8  ; Taping#1Conv'Fwd
      ANI     B0CA  ; Taping#1ConvStopSw
      AND     B0F31  ; Manual  ModeLampTaping
      LDI     M244  ; Taping#1Conv On At
      ANI     M252  ; Taping#1Conv On At
      INV
      ORB
      LD      Y0CC  ; U-BenderConv'Fwd
      ANI     Y0CE  ; U-BenderConv'   Slow
      LDI     Y0CC  ; U-BenderConv'Fwd
      OR      M244  ; Taping#1Conv On At
      ANI     X68E  ; Taping#1ConvWorkStop
      ORB
      ANB
      AND     X78  ; Buffer#2ConveyorConv' OLInv
      ANI     Y0C9  ; Taping#1Conv'Rev
      ANI     M6320  ; Buffer#2ConveyorConv' OLFault
      OUT     Y0C8  ; Taping#1Conv'Fwd
688   LD      B0C9  ; Taping#1Conv'RevSw
      ANI     B0CA  ; Taping#1ConvStopSw
      AND     B0F31  ; Manual  ModeLampTaping
      AND     X78  ; Buffer#2ConveyorConv' OLInv
      ANI     Y0C8  ; Taping#1Conv'Fwd
      ANI     M6320  ; Buffer#2ConveyorConv' OLFault
      OUT     Y0C9  ; Taping#1Conv'Rev
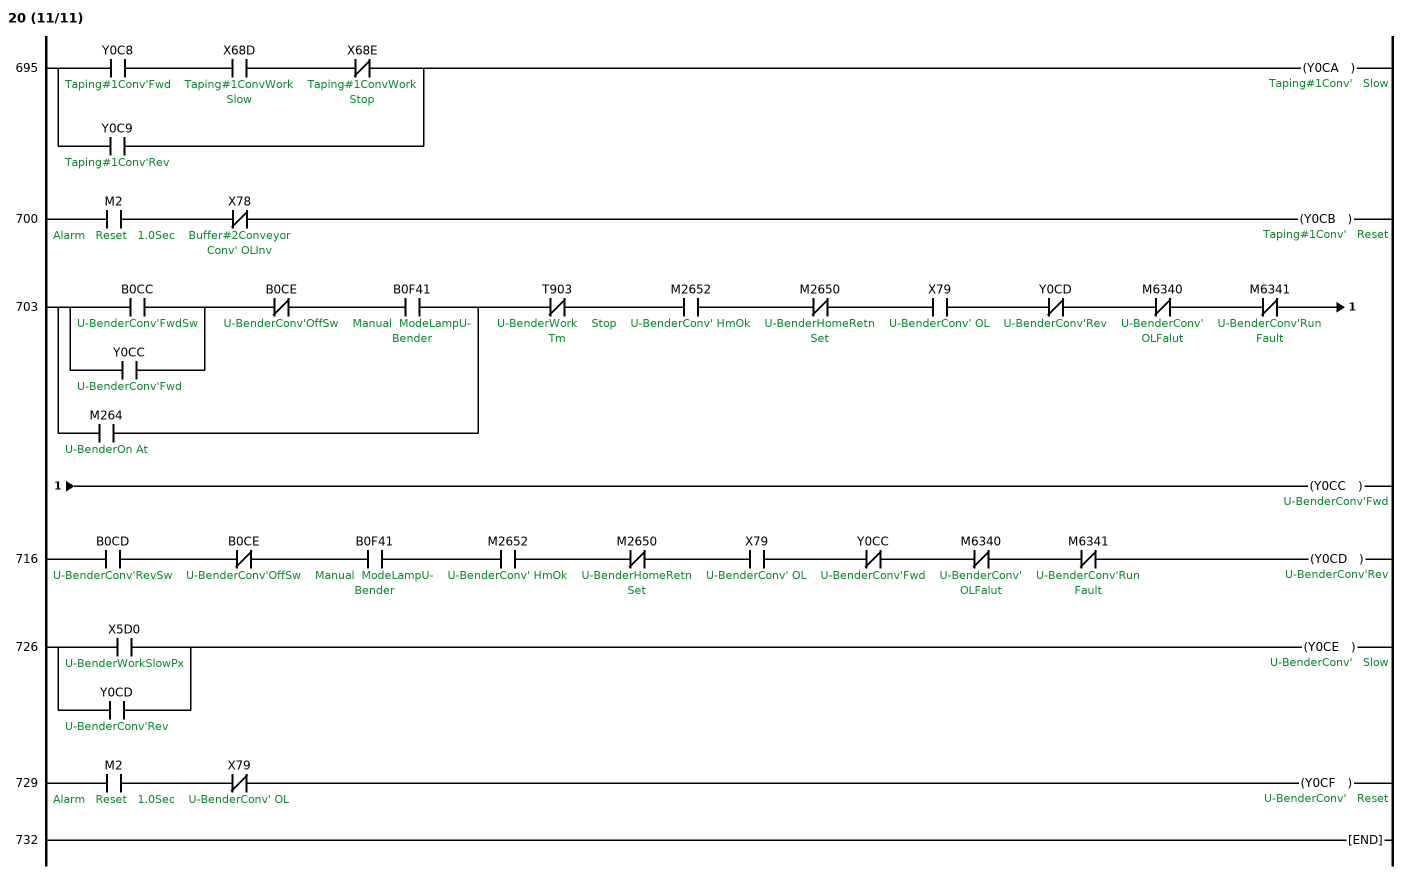
695   LD      Y0C8  ; Taping#1Conv'Fwd
      AND     X68D  ; Taping#1ConvWorkSlow
      ANI     X68E  ; Taping#1ConvWorkStop
      OR      Y0C9  ; Taping#1Conv'Rev
      OUT     Y0CA  ; Taping#1Conv'   Slow
700   LD      M2  ; Alarm   Reset   1.0Sec
      ANI     X78  ; Buffer#2ConveyorConv' OLInv
      OUT     Y0CB  ; Taping#1Conv'   Reset
703   LD      B0CC  ; U-BenderConv'FwdSw
      OR      Y0CC  ; U-BenderConv'Fwd
      ANI     B0CE  ; U-BenderConv'OffSw
      AND     B0F41  ; Manual  ModeLampU-Bender
      OR      M264  ; U-BenderOn At
      ANI     T903  ; U-BenderWork    Stop Tm
      AND     M2652  ; U-BenderConv' HmOk
      ANI     M2650  ; U-BenderHomeRetnSet
      AND     X79  ; U-BenderConv' OL
      ANI     Y0CD  ; U-BenderConv'Rev
      ANI     M6340  ; U-BenderConv' OLFalut
      ANI     M6341  ; U-BenderConv'RunFault
      OUT     Y0CC  ; U-BenderConv'Fwd
716   LD      B0CD  ; U-BenderConv'RevSw
      ANI     B0CE  ; U-BenderConv'OffSw
      AND     B0F41  ; Manual  ModeLampU-Bender
      AND     M2652  ; U-BenderConv' HmOk
      ANI     M2650  ; U-BenderHomeRetnSet
      AND     X79  ; U-BenderConv' OL
      ANI     Y0CC  ; U-BenderConv'Fwd
      ANI     M6340  ; U-BenderConv' OLFalut
      ANI     M6341  ; U-BenderConv'RunFault
      OUT     Y0CD  ; U-BenderConv'Rev
726   LD      X5D0  ; U-BenderWorkSlowPx
      OR      Y0CD  ; U-BenderConv'Rev
      OUT     Y0CE  ; U-BenderConv'   Slow
729   LD      M2  ; Alarm   Reset   1.0Sec
      ANI     X79  ; U-BenderConv' OL
      OUT     Y0CF  ; U-BenderConv'   Reset
732   END
END_PROGRAM

PROGRAM 21  // Divert Part
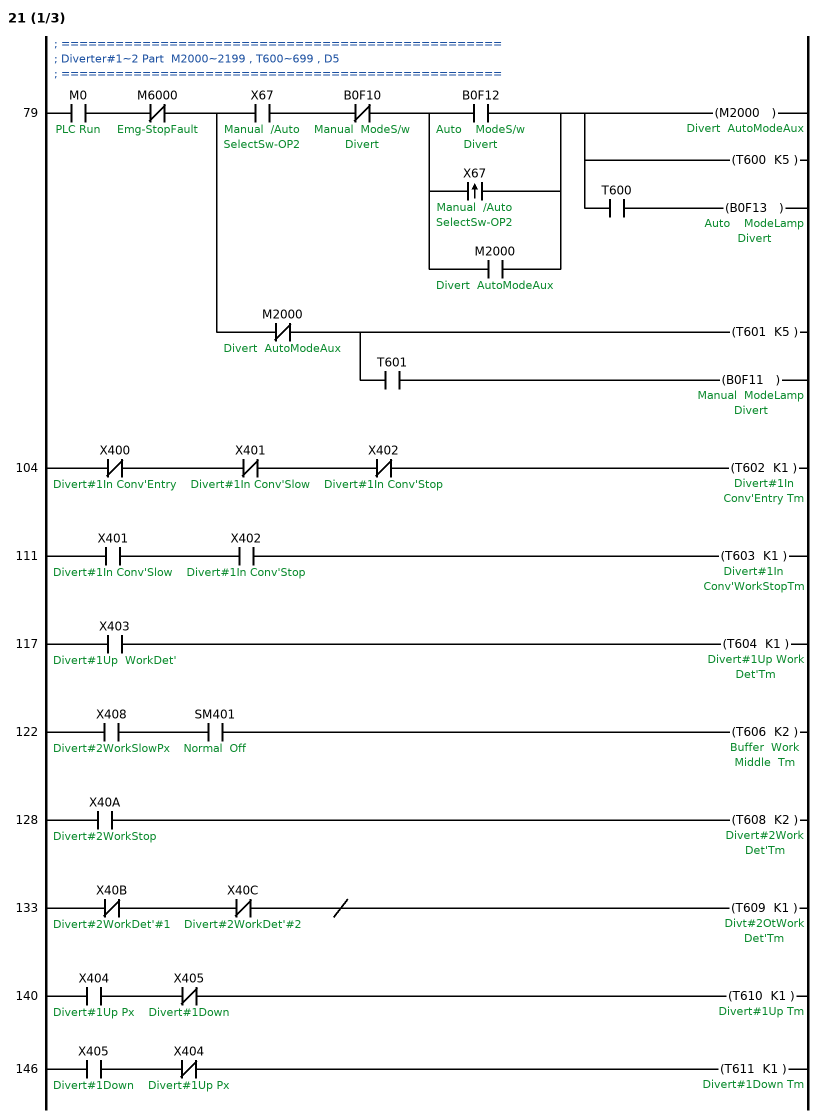
; =================================================
; Diverter#1~2 Part  M2000~2199 , T600~699 , D5
; =================================================
79    LD      M0  ; PLC Run
      ANI     M6000  ; Emg-StopFault
      MPS
      AND     X67  ; Manual  /Auto   SelectSw-OP2
      ANI     B0F10  ; Manual  ModeS/w Divert
      LD      B0F12  ; Auto    ModeS/w Divert
      ORP     X67  ; Manual  /Auto   SelectSw-OP2
      OR      M2000  ; Divert  AutoModeAux
      ANB
      OUT     M2000  ; Divert  AutoModeAux
      OUT     T600 K5
      AND     T600
      OUT     B0F13  ; Auto    ModeLampDivert
      MPP
      ANI     M2000  ; Divert  AutoModeAux
      OUT     T601 K5
      AND     T601
      OUT     B0F11  ; Manual  ModeLampDivert
104   LDI     X400  ; Divert#1In Conv'Entry
      ANI     X401  ; Divert#1In Conv'Slow
      ANI     X402  ; Divert#1In Conv'Stop
      OUT     T602 K1  ; Divert#1In Conv'Entry Tm
111   LD      X401  ; Divert#1In Conv'Slow
      AND     X402  ; Divert#1In Conv'Stop
      OUT     T603 K1  ; Divert#1In Conv'WorkStopTm
117   LD      X403  ; Divert#1Up  WorkDet'
      OUT     T604 K1  ; Divert#1Up Work Det'Tm
122   LD      X408  ; Divert#2WorkSlowPx
      AND     SM401  ; Normal  Off
      OUT     T606 K2  ; Buffer  Work    Middle  Tm
128   LD      X40A  ; Divert#2WorkStop
      OUT     T608 K2  ; Divert#2WorkDet'Tm
133   LDI     X40B  ; Divert#2WorkDet'#1
      ANI     X40C  ; Divert#2WorkDet'#2
      INV
      OUT     T609 K1  ; Divt#2OtWorkDet'Tm
140   LD      X404  ; Divert#1Up Px
      ANI     X405  ; Divert#1Down
      OUT     T610 K1  ; Divert#1Up Tm
146   LD      X405  ; Divert#1Down
      ANI     X404  ; Divert#1Up Px
      OUT     T611 K1  ; Divert#1Down Tm
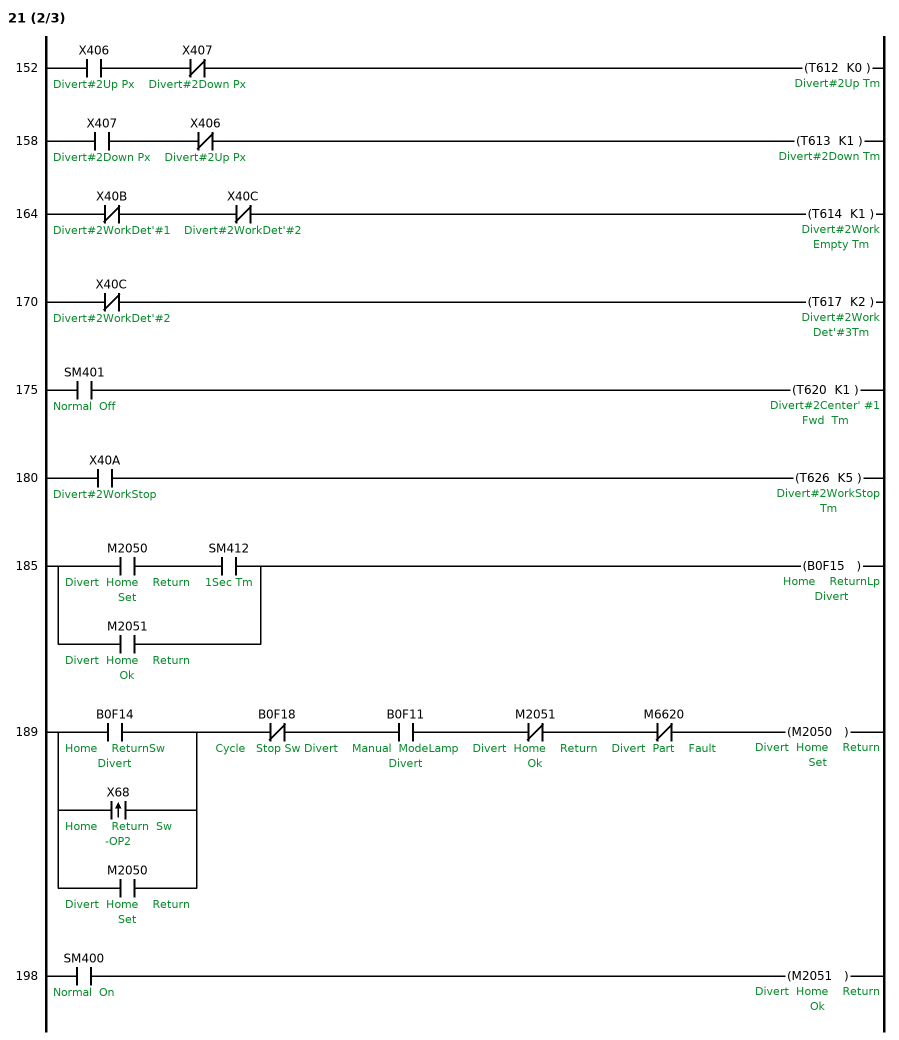
152   LD      X406  ; Divert#2Up Px
      ANI     X407  ; Divert#2Down Px
      OUT     T612 K0  ; Divert#2Up Tm
158   LD      X407  ; Divert#2Down Px
      ANI     X406  ; Divert#2Up Px
      OUT     T613 K1  ; Divert#2Down Tm
164   LDI     X40B  ; Divert#2WorkDet'#1
      ANI     X40C  ; Divert#2WorkDet'#2
      OUT     T614 K1  ; Divert#2Work    Empty Tm
170   LDI     X40C  ; Divert#2WorkDet'#2
      OUT     T617 K2  ; Divert#2WorkDet'#3Tm
175   LD      SM401  ; Normal  Off
      OUT     T620 K1  ; Divert#2Center' #1 Fwd  Tm
180   LD      X40A  ; Divert#2WorkStop
      OUT     T626 K5  ; Divert#2WorkStopTm
185   LD      M2050  ; Divert  Home    Return  Set
      AND     SM412  ; 1Sec Tm
      OR      M2051  ; Divert  Home    Return  Ok
      OUT     B0F15  ; Home    ReturnLpDivert
189   LD      B0F14  ; Home    ReturnSwDivert
      ORP     X68  ; Home    Return  Sw -OP2
      OR      M2050  ; Divert  Home    Return  Set
      ANI     B0F18  ; Cycle   Stop Sw Divert
      AND     B0F11  ; Manual  ModeLampDivert
      ANI     M2051  ; Divert  Home    Return  Ok
      ANI     M6620  ; Divert  Part    Fault
      OUT     M2050  ; Divert  Home    Return  Set
198   LD      SM400  ; Normal  On
      OUT     M2051  ; Divert  Home    Return  Ok
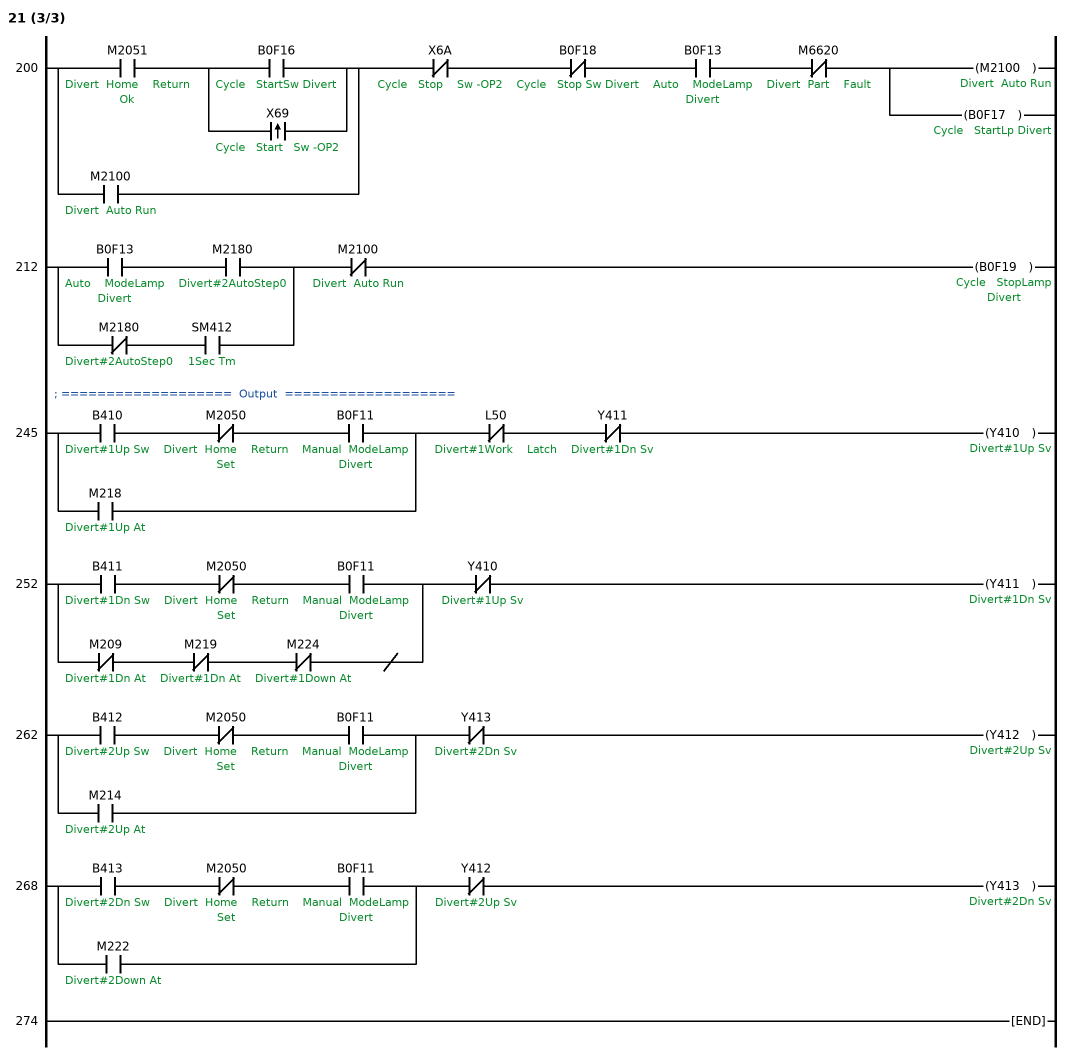
200   LD      M2051  ; Divert  Home    Return  Ok
      LD      B0F16  ; Cycle   StartSw Divert
      ORP     X69  ; Cycle   Start   Sw -OP2
      ANB
      OR      M2100  ; Divert  Auto Run
      ANI     X6A  ; Cycle   Stop    Sw -OP2
      ANI     B0F18  ; Cycle   Stop Sw Divert
      AND     B0F13  ; Auto    ModeLampDivert
      ANI     M6620  ; Divert  Part    Fault
      OUT     M2100  ; Divert  Auto Run
      OUT     B0F17  ; Cycle   StartLp Divert
212   LD      B0F13  ; Auto    ModeLampDivert
      AND     M2180  ; Divert#2AutoStep0
      LDI     M2180  ; Divert#2AutoStep0
      AND     SM412  ; 1Sec Tm
      ORB
      ANI     M2100  ; Divert  Auto Run
      OUT     B0F19  ; Cycle   StopLampDivert
; ===================  Output  ===================
245   LD      B410  ; Divert#1Up Sw
      ANI     M2050  ; Divert  Home    Return  Set
      AND     B0F11  ; Manual  ModeLampDivert
      OR      M218  ; Divert#1Up At
      ANI     L50  ; Divert#1Work    Latch
      ANI     Y411  ; Divert#1Dn Sv
      OUT     Y410  ; Divert#1Up Sv
252   LD      B411  ; Divert#1Dn Sw
      ANI     M2050  ; Divert  Home    Return  Set
      AND     B0F11  ; Manual  ModeLampDivert
      LDI     M209  ; Divert#1Dn At
      ANI     M219  ; Divert#1Dn At
      ANI     M224  ; Divert#1Down At
      INV
      ORB
      ANI     Y410  ; Divert#1Up Sv
      OUT     Y411  ; Divert#1Dn Sv
262   LD      B412  ; Divert#2Up Sw
      ANI     M2050  ; Divert  Home    Return  Set
      AND     B0F11  ; Manual  ModeLampDivert
      OR      M214  ; Divert#2Up At
      ANI     Y413  ; Divert#2Dn Sv
      OUT     Y412  ; Divert#2Up Sv
268   LD      B413  ; Divert#2Dn Sw
      ANI     M2050  ; Divert  Home    Return  Set
      AND     B0F11  ; Manual  ModeLampDivert
      OR      M222  ; Divert#2Down At
      ANI     Y412  ; Divert#2Up Sv
      OUT     Y413  ; Divert#2Dn Sv
274   END
END_PROGRAM

PROGRAM 22  // L-Bender(Z)
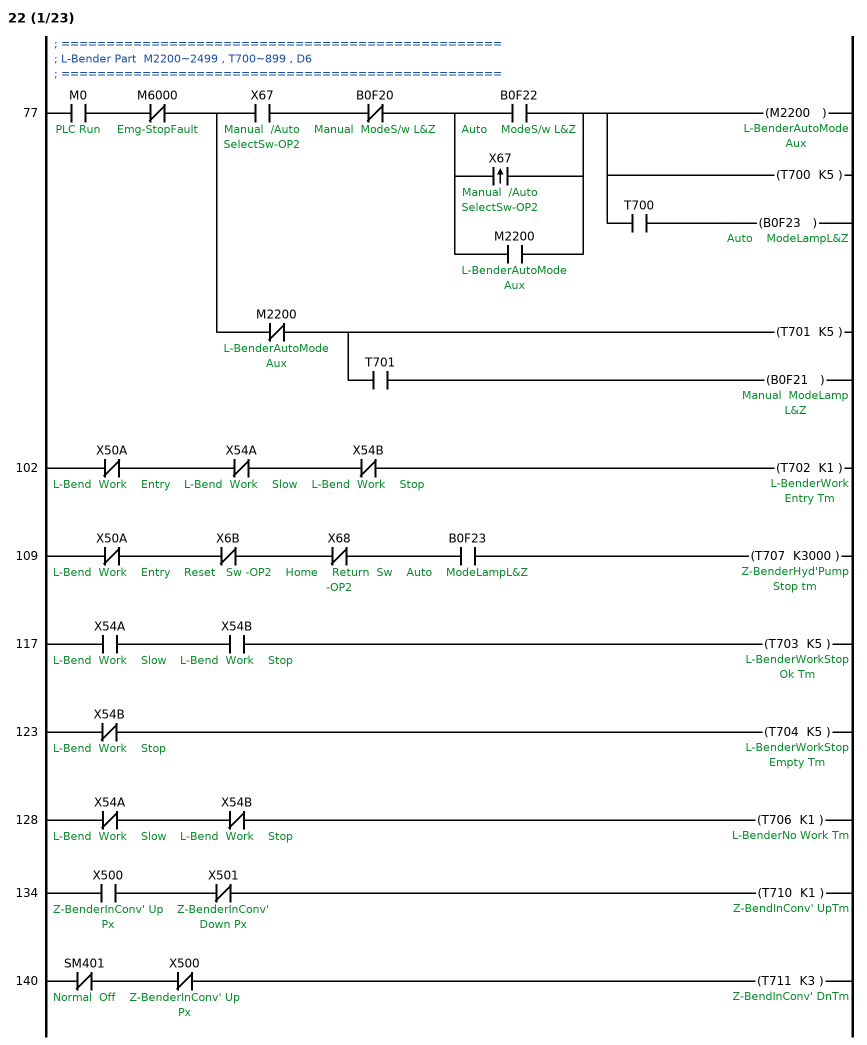
; =================================================
; L-Bender Part  M2200~2499 , T700~899 , D6
; =================================================
77    LD      M0  ; PLC Run
      ANI     M6000  ; Emg-StopFault
      MPS
      AND     X67  ; Manual  /Auto   SelectSw-OP2
      ANI     B0F20  ; Manual  ModeS/w L&Z
      LD      B0F22  ; Auto    ModeS/w L&Z
      ORP     X67  ; Manual  /Auto   SelectSw-OP2
      OR      M2200  ; L-BenderAutoModeAux
      ANB
      OUT     M2200  ; L-BenderAutoModeAux
      OUT     T700 K5
      AND     T700
      OUT     B0F23  ; Auto    ModeLampL&Z
      MPP
      ANI     M2200  ; L-BenderAutoModeAux
      OUT     T701 K5
      AND     T701
      OUT     B0F21  ; Manual  ModeLampL&Z
102   LDI     X50A  ; L-Bend  Work    Entry
      ANI     X54A  ; L-Bend  Work    Slow
      ANI     X54B  ; L-Bend  Work    Stop
      OUT     T702 K1  ; L-BenderWork    Entry Tm
109   LDI     X50A  ; L-Bend  Work    Entry
      ANI     X6B  ; Reset   Sw -OP2
      ANI     X68  ; Home    Return  Sw -OP2
      AND     B0F23  ; Auto    ModeLampL&Z
      OUT     T707 K3000  ; Z-BenderHyd'PumpStop tm
117   LD      X54A  ; L-Bend  Work    Slow
      AND     X54B  ; L-Bend  Work    Stop
      OUT     T703 K5  ; L-BenderWorkStopOk Tm
123   LDI     X54B  ; L-Bend  Work    Stop
      OUT     T704 K5  ; L-BenderWorkStopEmpty Tm
128   LDI     X54A  ; L-Bend  Work    Slow
      ANI     X54B  ; L-Bend  Work    Stop
      OUT     T706 K1  ; L-BenderNo Work Tm
134   LD      X500  ; Z-BenderInConv' Up Px
      ANI     X501  ; Z-BenderInConv' Down Px
      OUT     T710 K1  ; Z-BendInConv' UpTm
140   LDI     SM401  ; Normal  Off
      ANI     X500  ; Z-BenderInConv' Up Px
      OUT     T711 K3  ; Z-BendInConv' DnTm
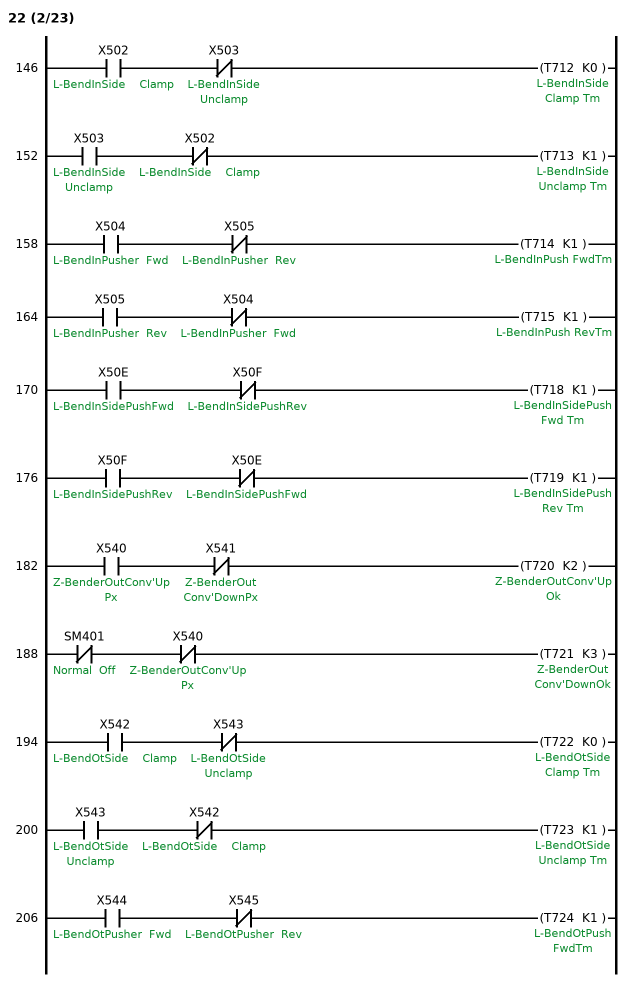
146   LD      X502  ; L-BendInSide    Clamp
      ANI     X503  ; L-BendInSide    Unclamp
      OUT     T712 K0  ; L-BendInSide    Clamp Tm
152   LD      X503  ; L-BendInSide    Unclamp
      ANI     X502  ; L-BendInSide    Clamp
      OUT     T713 K1  ; L-BendInSide    Unclamp Tm
158   LD      X504  ; L-BendInPusher  Fwd
      ANI     X505  ; L-BendInPusher  Rev
      OUT     T714 K1  ; L-BendInPush FwdTm
164   LD      X505  ; L-BendInPusher  Rev
      ANI     X504  ; L-BendInPusher  Fwd
      OUT     T715 K1  ; L-BendInPush RevTm
170   LD      X50E  ; L-BendInSidePushFwd
      ANI     X50F  ; L-BendInSidePushRev
      OUT     T718 K1  ; L-BendInSidePushFwd Tm
176   LD      X50F  ; L-BendInSidePushRev
      ANI     X50E  ; L-BendInSidePushFwd
      OUT     T719 K1  ; L-BendInSidePushRev Tm
182   LD      X540  ; Z-BenderOutConv'Up Px
      ANI     X541  ; Z-BenderOutConv'DownPx
      OUT     T720 K2  ; Z-BenderOutConv'Up Ok
188   LDI     SM401  ; Normal  Off
      ANI     X540  ; Z-BenderOutConv'Up Px
      OUT     T721 K3  ; Z-BenderOutConv'DownOk
194   LD      X542  ; L-BendOtSide    Clamp
      ANI     X543  ; L-BendOtSide    Unclamp
      OUT     T722 K0  ; L-BendOtSide    Clamp Tm
200   LD      X543  ; L-BendOtSide    Unclamp
      ANI     X542  ; L-BendOtSide    Clamp
      OUT     T723 K1  ; L-BendOtSide    Unclamp Tm
206   LD      X544  ; L-BendOtPusher  Fwd
      ANI     X545  ; L-BendOtPusher  Rev
      OUT     T724 K1  ; L-BendOtPush FwdTm
